Yaskawa INFORM job: DEMO_ROOF_UPPER_0625_3PAINT_54.JBI

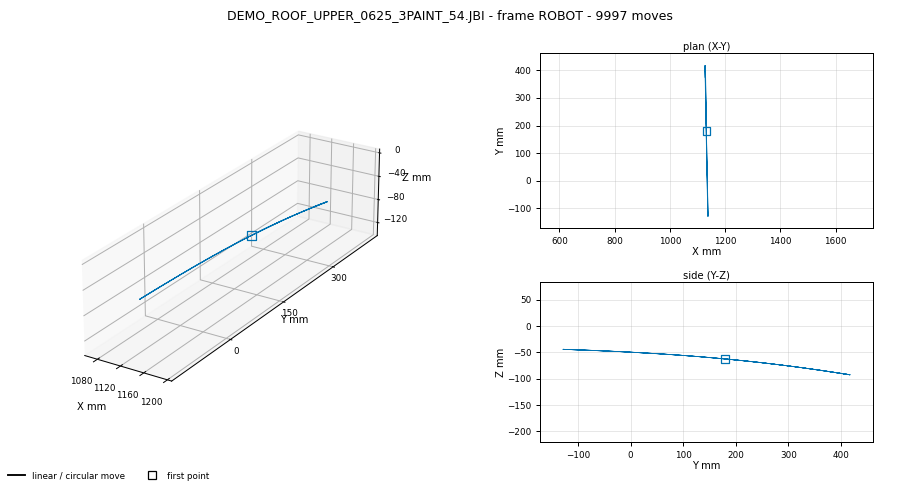
[picture p0: tool path of DEMO_ROOF_UPPER_0625_3PAINT_54.JBI in frame ROBOT, 9997 of 9997 moves have a stored position in this frame; points joined in program order, loops and branches not executed]
/JOB
//NAME DEMO_ROOF_UPPER_0625_3PAINT54
//POS
///NPOS 9997,0,0,0,0,0
///TOOL 0
///USER 0
///POSTYPE ROBOT
///RECTAN
///RCONF 1,0,0,0,0,0,0,0,0,0,0,0,0,0,0,0,0,0,0,0,0,0,0,0
C00000=1132.643,178.804,-62.011,-179.310,9.058,149.575
C00001=1132.639,179.053,-62.034,-179.309,9.060,149.575
C00002=1132.634,179.302,-62.058,-179.306,9.063,149.575
C00003=1132.629,179.551,-62.081,-179.303,9.067,149.575
C00004=1132.624,179.799,-62.104,-179.299,9.071,149.575
C00005=1132.620,180.048,-62.127,-179.296,9.074,149.575
C00006=1132.615,180.297,-62.150,-179.293,9.077,149.575
C00007=1132.611,180.546,-62.174,-179.290,9.081,149.575
C00008=1132.606,180.795,-62.198,-179.287,9.085,149.575
C00009=1132.602,181.044,-62.221,-179.284,9.088,149.575
C00010=1132.597,181.293,-62.244,-179.281,9.092,149.575
C00011=1132.592,181.541,-62.268,-179.278,9.094,149.575
C00012=1132.588,181.790,-62.292,-179.275,9.098,149.575
C00013=1132.583,182.039,-62.315,-179.272,9.101,149.575
C00014=1132.579,182.288,-62.339,-179.268,9.105,149.575
C00015=1132.574,182.537,-62.363,-179.266,9.108,149.575
C00016=1132.569,182.786,-62.386,-179.263,9.111,149.575
C00017=1132.565,183.035,-62.410,-179.260,9.114,149.575
C00018=1132.561,183.284,-62.434,-179.257,9.118,149.575
C00019=1132.556,183.533,-62.457,-179.254,9.120,149.575
C00020=1132.552,183.781,-62.481,-179.251,9.124,149.575
C00021=1132.547,184.030,-62.505,-179.249,9.127,149.575
C00022=1132.542,184.279,-62.528,-179.246,9.130,149.575
C00023=1132.538,184.494,-62.549,-179.244,9.132,149.575
C00024=1132.535,184.707,-62.569,-179.241,9.135,149.575
C00025=1132.531,184.922,-62.589,-179.239,9.138,149.575
C00026=1132.527,185.137,-62.610,-179.237,9.141,149.575
C00027=1132.523,185.351,-62.631,-179.235,9.143,149.575
C00028=1132.519,185.566,-62.651,-179.232,9.146,149.575
C00029=1132.515,185.781,-62.672,-179.230,9.148,149.575
C00030=1132.512,185.995,-62.692,-179.228,9.151,149.575
C00031=1132.506,186.244,-62.716,-179.226,9.154,149.575
C00032=1132.502,186.493,-62.740,-179.223,9.157,149.575
C00033=1132.497,186.741,-62.764,-179.221,9.160,149.575
C00034=1132.493,186.990,-62.787,-179.218,9.163,149.575
C00035=1132.488,187.239,-62.811,-179.215,9.166,149.575
C00036=1132.484,187.487,-62.835,-179.213,9.168,149.575
C00037=1132.479,187.736,-62.859,-179.211,9.171,149.575
C00038=1132.475,187.986,-62.884,-179.208,9.174,149.575
C00039=1132.470,188.235,-62.907,-179.206,9.177,149.575
C00040=1132.466,188.483,-62.931,-179.204,9.180,149.575
C00041=1132.461,188.732,-62.955,-179.202,9.182,149.575
C00042=1132.456,188.981,-62.979,-179.199,9.185,149.575
C00043=1132.451,189.229,-63.003,-179.197,9.188,149.575
C00044=1132.447,189.478,-63.027,-179.195,9.191,149.575
C00045=1132.443,189.727,-63.051,-179.193,9.193,149.575
C00046=1132.438,189.976,-63.075,-179.191,9.196,149.575
C00047=1132.434,190.224,-63.099,-179.189,9.199,149.575
C00048=1132.429,190.474,-63.123,-179.187,9.202,149.575
C00049=1132.424,190.722,-63.147,-179.185,9.204,149.575
C00050=1132.420,190.971,-63.172,-179.183,9.207,149.575
C00051=1132.415,191.220,-63.196,-179.181,9.210,149.576
C00052=1132.411,191.469,-63.220,-179.179,9.212,149.576
C00053=1132.406,191.717,-63.244,-179.177,9.215,149.576
C00054=1132.402,191.966,-63.268,-179.175,9.217,149.576
C00055=1132.397,192.215,-63.293,-179.174,9.220,149.576
C00056=1132.393,192.464,-63.317,-179.172,9.222,149.576
C00057=1132.388,192.713,-63.340,-179.170,9.226,149.576
C00058=1132.383,192.961,-63.365,-179.168,9.228,149.576
C00059=1132.379,193.210,-63.389,-179.166,9.231,149.577
C00060=1132.375,193.459,-63.414,-179.164,9.233,149.577
C00061=1132.370,193.708,-63.438,-179.163,9.236,149.577
C00062=1132.365,193.956,-63.462,-179.161,9.238,149.577
C00063=1132.361,194.205,-63.486,-179.160,9.240,149.577
C00064=1132.356,194.454,-63.511,-179.158,9.242,149.577
C00065=1132.352,194.703,-63.535,-179.157,9.245,149.577
C00066=1132.347,194.951,-63.559,-179.155,9.248,149.578
C00067=1132.343,195.201,-63.584,-179.153,9.250,149.578
C00068=1132.338,195.449,-63.608,-179.152,9.253,149.578
C00069=1132.334,195.698,-63.632,-179.151,9.255,149.578
C00070=1132.329,195.946,-63.657,-179.150,9.257,149.578
C00071=1132.325,196.195,-63.681,-179.148,9.260,149.579
C00072=1132.320,196.444,-63.706,-179.145,9.263,149.578
C00073=1132.316,196.692,-63.730,-179.140,9.268,149.578
C00074=1132.312,196.942,-63.754,-179.136,9.272,149.578
C00075=1132.307,197.190,-63.779,-179.132,9.275,149.578
C00076=1132.302,197.439,-63.803,-179.128,9.279,149.578
C00077=1132.297,197.687,-63.828,-179.124,9.284,149.578
C00078=1132.293,197.937,-63.852,-179.120,9.287,149.577
C00079=1132.289,198.151,-63.873,-179.116,9.291,149.577
C00080=1132.285,198.365,-63.895,-179.112,9.294,149.577
C00081=1132.281,198.580,-63.916,-179.109,9.297,149.577
C00082=1132.277,198.795,-63.937,-179.106,9.300,149.577
C00083=1132.274,199.009,-63.958,-179.103,9.303,149.576
C00084=1132.270,199.223,-63.979,-179.099,9.306,149.576
C00085=1132.265,199.437,-64.001,-179.096,9.309,149.576
C00086=1132.261,199.652,-64.022,-179.093,9.313,149.576
C00087=1132.258,199.901,-64.047,-179.089,9.316,149.576
C00088=1132.253,200.149,-64.071,-179.086,9.320,149.576
C00089=1132.248,200.399,-64.096,-179.082,9.323,149.576
C00090=1132.244,200.647,-64.121,-179.078,9.327,149.576
C00091=1132.239,200.895,-64.146,-179.075,9.330,149.575
C00092=1132.235,201.144,-64.170,-179.071,9.334,149.575
C00093=1132.230,201.393,-64.195,-179.068,9.336,149.575
C00094=1132.226,201.642,-64.221,-179.064,9.340,149.575
C00095=1132.221,201.890,-64.245,-179.061,9.343,149.575
C00096=1132.217,202.140,-64.270,-179.058,9.346,149.574
C00097=1132.212,202.388,-64.295,-179.054,9.349,149.574
C00098=1132.208,202.637,-64.320,-179.051,9.353,149.574
C00099=1132.203,202.886,-64.344,-179.048,9.356,149.574
C00100=1132.199,203.134,-64.370,-179.045,9.358,149.574
C00101=1132.195,203.383,-64.394,-179.041,9.362,149.574
C00102=1132.190,203.632,-64.420,-179.039,9.365,149.574
C00103=1132.185,203.880,-64.445,-179.036,9.368,149.574
C00104=1132.181,204.129,-64.470,-179.032,9.371,149.574
C00105=1132.177,204.378,-64.494,-179.029,9.374,149.573
C00106=1132.172,204.626,-64.520,-179.026,9.377,149.573
C00107=1132.167,204.875,-64.545,-179.023,9.379,149.573
C00108=1132.163,205.124,-64.571,-179.021,9.383,149.573
C00109=1132.159,205.372,-64.595,-179.018,9.385,149.573
C00110=1132.154,205.621,-64.620,-179.015,9.388,149.573
C00111=1132.149,205.870,-64.645,-179.012,9.391,149.573
C00112=1132.145,206.119,-64.671,-179.009,9.394,149.573
C00113=1132.140,206.367,-64.696,-179.006,9.397,149.573
C00114=1132.136,206.616,-64.721,-179.004,9.400,149.573
C00115=1132.132,206.864,-64.746,-179.002,9.402,149.572
C00116=1132.127,207.113,-64.772,-178.999,9.405,149.573
C00117=1132.123,207.362,-64.797,-178.996,9.408,149.573
C00118=1132.118,207.610,-64.822,-178.994,9.410,149.572
C00119=1132.114,207.859,-64.848,-178.992,9.413,149.572
C00120=1132.109,208.108,-64.873,-178.990,9.415,149.573
C00121=1132.104,208.357,-64.898,-178.987,9.418,149.572
C00122=1132.100,208.605,-64.924,-178.985,9.420,149.572
C00123=1132.096,208.854,-64.948,-178.982,9.424,149.572
C00124=1132.092,209.103,-64.974,-178.980,9.426,149.573
C00125=1132.087,209.351,-64.999,-178.979,9.428,149.573
C00126=1132.083,209.600,-65.025,-178.976,9.431,149.573
C00127=1132.078,209.849,-65.050,-178.974,9.434,149.573
C00128=1132.073,210.097,-65.076,-178.972,9.436,149.573
C00129=1132.069,210.346,-65.101,-178.970,9.438,149.573
C00130=1132.065,210.595,-65.127,-178.968,9.441,149.573
C00131=1132.060,210.843,-65.152,-178.967,9.443,149.573
C00132=1132.055,211.092,-65.178,-178.965,9.446,149.573
C00133=1132.051,211.340,-65.203,-178.963,9.448,149.573
C00134=1132.046,211.589,-65.229,-178.961,9.450,149.573
C00135=1132.043,211.803,-65.250,-178.960,9.453,149.573
C00136=1132.039,212.018,-65.273,-178.959,9.455,149.573
C00137=1132.035,212.232,-65.295,-178.957,9.457,149.573
C00138=1132.031,212.446,-65.316,-178.956,9.459,149.574
C00139=1132.027,212.661,-65.338,-178.954,9.462,149.574
C00140=1132.024,212.875,-65.361,-178.953,9.463,149.574
C00141=1132.020,213.089,-65.383,-178.952,9.465,149.574
C00142=1132.015,213.303,-65.405,-178.950,9.467,149.574
C00143=1132.011,213.552,-65.431,-178.949,9.470,149.574
C00144=1132.007,213.801,-65.456,-178.947,9.473,149.575
C00145=1132.002,214.049,-65.482,-178.946,9.475,149.575
C00146=1131.998,214.298,-65.508,-178.944,9.478,149.575
C00147=1131.993,214.547,-65.533,-178.942,9.480,149.575
C00148=1131.989,214.796,-65.558,-178.940,9.484,149.575
C00149=1131.984,215.044,-65.584,-178.938,9.486,149.575
C00150=1131.980,215.293,-65.609,-178.937,9.489,149.576
C00151=1131.976,215.542,-65.635,-178.934,9.492,149.576
C00152=1131.971,215.790,-65.661,-178.933,9.494,149.576
C00153=1131.967,216.039,-65.686,-178.931,9.497,149.576
C00154=1131.962,216.287,-65.712,-178.929,9.500,149.576
C00155=1131.958,216.536,-65.738,-178.927,9.503,149.576
C00156=1131.953,216.784,-65.765,-178.924,9.506,149.576
C00157=1131.949,217.033,-65.790,-178.922,9.509,149.577
C00158=1131.945,217.282,-65.816,-178.920,9.511,149.577
C00159=1131.940,217.530,-65.842,-178.918,9.515,149.577
C00160=1131.935,217.778,-65.867,-178.916,9.518,149.577
C00161=1131.931,218.027,-65.893,-178.914,9.520,149.577
C00162=1131.927,218.276,-65.919,-178.911,9.523,149.577
C00163=1131.922,218.525,-65.945,-178.909,9.527,149.577
C00164=1131.917,218.773,-65.970,-178.907,9.530,149.577
C00165=1131.913,219.022,-65.996,-178.905,9.532,149.577
C00166=1131.909,219.270,-66.023,-178.902,9.535,149.577
C00167=1131.905,219.519,-66.048,-178.900,9.539,149.578
C00168=1131.901,219.768,-66.074,-178.897,9.542,149.578
C00169=1131.895,220.016,-66.100,-178.895,9.545,149.578
C00170=1131.891,220.265,-66.126,-178.892,9.548,149.578
C00171=1131.887,220.513,-66.152,-178.890,9.551,149.578
C00172=1131.883,220.762,-66.178,-178.887,9.554,149.578
C00173=1131.878,221.011,-66.204,-178.884,9.558,149.578
C00174=1131.874,221.260,-66.230,-178.881,9.561,149.578
C00175=1131.869,221.508,-66.256,-178.879,9.564,149.578
C00176=1131.865,221.756,-66.282,-178.876,9.567,149.578
C00177=1131.860,222.005,-66.308,-178.874,9.570,149.578
C00178=1131.856,222.254,-66.335,-178.871,9.574,149.578
C00179=1131.852,222.502,-66.361,-178.868,9.577,149.578
C00180=1131.847,222.752,-66.387,-178.865,9.580,149.578
C00181=1131.843,223.000,-66.413,-178.862,9.584,149.578
C00182=1131.838,223.248,-66.439,-178.859,9.587,149.578
C00183=1131.833,223.497,-66.465,-178.856,9.591,149.578
C00184=1131.829,223.745,-66.492,-178.853,9.594,149.578
C00185=1131.825,223.994,-66.517,-178.850,9.598,149.578
C00186=1131.820,224.242,-66.544,-178.847,9.600,149.578
C00187=1131.816,224.491,-66.570,-178.844,9.604,149.578
C00188=1131.811,224.740,-66.597,-178.840,9.608,149.578
C00189=1131.807,224.989,-66.623,-178.838,9.611,149.578
C00190=1131.803,225.237,-66.649,-178.834,9.614,149.578
C00191=1131.799,225.451,-66.672,-178.832,9.618,149.578
C00192=1131.795,225.665,-66.695,-178.829,9.620,149.578
C00193=1131.791,225.879,-66.717,-178.826,9.623,149.578
C00194=1131.788,226.094,-66.740,-178.823,9.626,149.578
C00195=1131.784,226.308,-66.763,-178.820,9.629,149.578
C00196=1131.780,226.522,-66.786,-178.817,9.633,149.578
C00197=1131.776,226.736,-66.809,-178.814,9.636,149.578
C00198=1131.772,226.951,-66.831,-178.811,9.638,149.578
C00199=1131.768,227.199,-66.858,-178.808,9.642,149.578
C00200=1131.764,227.447,-66.885,-178.804,9.645,149.577
C00201=1131.759,227.696,-66.911,-178.801,9.649,149.577
C00202=1131.755,227.945,-66.937,-178.797,9.652,149.577
C00203=1131.750,228.193,-66.964,-178.793,9.656,149.577
C00204=1131.746,228.441,-66.991,-178.790,9.659,149.577
C00205=1131.741,228.690,-67.017,-178.786,9.663,149.577
C00206=1131.737,228.939,-67.044,-178.783,9.666,149.577
C00207=1131.733,229.187,-67.071,-178.779,9.670,149.577
C00208=1131.728,229.436,-67.098,-178.775,9.673,149.576
C00209=1131.724,229.684,-67.124,-178.771,9.677,149.576
C00210=1131.719,229.933,-67.151,-178.767,9.681,149.576
C00211=1131.715,230.181,-67.178,-178.763,9.684,149.576
C00212=1131.711,230.430,-67.204,-178.760,9.688,149.576
C00213=1131.706,230.678,-67.231,-178.756,9.691,149.576
C00214=1131.701,230.927,-67.258,-178.752,9.694,149.575
C00215=1131.697,231.175,-67.285,-178.749,9.698,149.575
C00216=1131.693,231.423,-67.312,-178.745,9.701,149.575
C00217=1131.688,231.672,-67.339,-178.741,9.704,149.575
C00218=1131.684,231.921,-67.365,-178.737,9.708,149.575
C00219=1131.680,232.170,-67.392,-178.734,9.711,149.574
C00220=1131.675,232.418,-67.419,-178.731,9.714,149.574
C00221=1131.670,232.667,-67.446,-178.727,9.718,149.574
C00222=1131.667,232.915,-67.473,-178.724,9.720,149.574
C00223=1131.662,233.163,-67.500,-178.720,9.724,149.574
C00224=1131.658,233.411,-67.528,-178.717,9.726,149.574
C00225=1131.654,233.660,-67.555,-178.714,9.729,149.573
C00226=1131.650,233.909,-67.581,-178.711,9.733,149.573
C00227=1131.645,234.157,-67.609,-178.708,9.735,149.573
C00228=1131.640,234.406,-67.636,-178.705,9.738,149.573
C00229=1131.636,234.654,-67.663,-178.701,9.741,149.573
C00230=1131.631,234.903,-67.690,-178.698,9.744,149.573
C00231=1131.627,235.152,-67.717,-178.695,9.747,149.573
C00232=1131.623,235.399,-67.744,-178.692,9.750,149.572
C00233=1131.619,235.648,-67.771,-178.689,9.752,149.572
C00234=1131.614,235.896,-67.798,-178.686,9.755,149.572
C00235=1131.610,236.146,-67.826,-178.683,9.758,149.572
C00236=1131.605,236.394,-67.853,-178.680,9.761,149.572
C00237=1131.601,236.642,-67.881,-178.678,9.764,149.572
C00238=1131.596,236.890,-67.908,-178.675,9.766,149.572
C00239=1131.592,237.139,-67.935,-178.672,9.769,149.572
C00240=1131.589,237.387,-67.962,-178.670,9.771,149.572
C00241=1131.584,237.636,-67.989,-178.667,9.774,149.571
C00242=1131.579,237.884,-68.016,-178.664,9.777,149.571
C00243=1131.575,238.133,-68.044,-178.662,9.779,149.571
C00244=1131.571,238.381,-68.072,-178.659,9.782,149.571
C00245=1131.566,238.630,-68.099,-178.657,9.784,149.571
C00246=1131.562,238.878,-68.126,-178.654,9.787,149.571
C00247=1131.558,239.092,-68.150,-178.652,9.789,149.571
C00248=1131.554,239.307,-68.173,-178.650,9.791,149.571
C00249=1131.551,239.520,-68.197,-178.647,9.793,149.571
C00250=1131.546,239.734,-68.221,-178.646,9.795,149.571
C00251=1131.543,239.948,-68.245,-178.644,9.797,149.571
C00252=1131.539,240.163,-68.268,-178.642,9.799,149.571
C00253=1131.536,240.377,-68.292,-178.640,9.801,149.571
C00254=1131.531,240.590,-68.316,-178.638,9.803,149.571
C00255=1131.527,240.839,-68.344,-178.636,9.806,149.571
C00256=1131.523,241.088,-68.371,-178.634,9.808,149.571
C00257=1131.518,241.335,-68.399,-178.632,9.810,149.571
C00258=1131.514,241.585,-68.426,-178.630,9.812,149.571
C00259=1131.510,241.832,-68.454,-178.628,9.815,149.571
C00260=1131.505,242.081,-68.481,-178.626,9.817,149.571
C00261=1131.502,242.330,-68.509,-178.624,9.819,149.571
C00262=1131.497,242.578,-68.536,-178.622,9.821,149.571
C00263=1131.493,242.826,-68.564,-178.620,9.824,149.571
C00264=1131.488,243.075,-68.591,-178.618,9.826,149.571
C00265=1131.484,243.323,-68.619,-178.617,9.827,149.571
C00266=1131.479,243.572,-68.646,-178.615,9.830,149.571
C00267=1131.476,243.820,-68.674,-178.613,9.832,149.571
C00268=1131.470,244.069,-68.702,-178.611,9.835,149.571
C00269=1131.466,244.317,-68.730,-178.610,9.836,149.571
C00270=1131.462,244.565,-68.758,-178.608,9.839,149.572
C00271=1131.458,244.814,-68.785,-178.607,9.841,149.572
C00272=1131.454,245.062,-68.813,-178.606,9.843,149.572
C00273=1131.449,245.311,-68.840,-178.604,9.844,149.572
C00274=1131.445,245.559,-68.868,-178.603,9.847,149.572
C00275=1131.441,245.807,-68.896,-178.602,9.849,149.572
C00276=1131.436,246.056,-68.924,-178.601,9.851,149.572
C00277=1131.431,246.304,-68.951,-178.599,9.853,149.573
C00278=1131.428,246.553,-68.980,-178.598,9.855,149.573
C00279=1131.423,246.801,-69.007,-178.597,9.857,149.573
C00280=1131.419,247.050,-69.035,-178.596,9.859,149.573
C00281=1131.415,247.298,-69.063,-178.595,9.861,149.573
C00282=1131.409,247.546,-69.090,-178.590,9.865,149.573
C00283=1131.406,247.795,-69.118,-178.583,9.871,149.573
C00284=1131.401,248.043,-69.146,-178.575,9.876,149.572
C00285=1131.398,248.291,-69.174,-178.568,9.882,149.571
C00286=1131.392,248.540,-69.202,-178.561,9.888,149.571
C00287=1131.388,248.789,-69.230,-178.554,9.893,149.570
C00288=1131.384,249.037,-69.258,-178.548,9.897,149.570
C00289=1131.380,249.286,-69.287,-178.542,9.902,149.569
C00290=1131.375,249.533,-69.314,-178.536,9.906,149.569
C00291=1131.371,249.782,-69.342,-178.531,9.911,149.568
C00292=1131.366,250.030,-69.371,-178.526,9.914,149.568
C00293=1131.363,250.279,-69.399,-178.520,9.919,149.567
C00294=1131.358,250.527,-69.427,-178.516,9.922,149.567
C00295=1131.354,250.776,-69.456,-178.511,9.925,149.567
C00296=1131.349,251.023,-69.483,-178.507,9.928,149.566
C00297=1131.345,251.272,-69.512,-178.503,9.932,149.566
C00298=1131.341,251.520,-69.540,-178.499,9.935,149.566
C00299=1131.337,251.769,-69.568,-178.496,9.938,149.566
C00300=1131.332,252.018,-69.597,-178.493,9.940,149.565
C00301=1131.328,252.266,-69.624,-178.490,9.943,149.565
C00302=1131.324,252.514,-69.654,-178.487,9.945,149.565
C00303=1131.320,252.728,-69.678,-178.485,9.947,149.565
C00304=1131.316,252.942,-69.703,-178.483,9.949,149.565
C00305=1131.313,253.156,-69.727,-178.482,9.950,149.565
C00306=1131.309,253.370,-69.751,-178.480,9.952,149.565
C00307=1131.305,253.584,-69.776,-178.479,9.953,149.565
C00308=1131.301,253.798,-69.800,-178.477,9.954,149.565
C00309=1131.298,254.011,-69.825,-178.477,9.956,149.565
C00310=1131.294,254.225,-69.850,-178.476,9.956,149.565
C00311=1131.290,254.473,-69.878,-178.476,9.958,149.565
C00312=1131.285,254.722,-69.906,-178.475,9.959,149.565
C00313=1131.281,254.971,-69.934,-178.476,9.960,149.566
C00314=1131.277,255.218,-69.963,-178.476,9.960,149.566
C00315=1131.273,255.467,-69.992,-178.476,9.962,149.566
C00316=1131.268,255.716,-70.020,-178.478,9.962,149.567
C00317=1131.264,255.963,-70.048,-178.479,9.962,149.567
C00318=1131.259,256.212,-70.077,-178.476,9.965,149.567
C00319=1131.255,256.460,-70.105,-178.473,9.968,149.567
C00320=1131.251,256.708,-70.134,-178.469,9.971,149.567
C00321=1131.247,256.957,-70.162,-178.466,9.974,149.567
C00322=1131.242,257.205,-70.191,-178.463,9.977,149.566
C00323=1131.238,257.454,-70.220,-178.460,9.980,149.566
C00324=1131.234,257.702,-70.248,-178.457,9.982,149.566
C00325=1131.229,257.950,-70.277,-178.455,9.985,149.566
C00326=1131.226,258.198,-70.305,-178.451,9.989,149.566
C00327=1131.221,258.447,-70.334,-178.448,9.991,149.566
C00328=1131.216,258.695,-70.363,-178.445,9.994,149.566
C00329=1131.213,258.943,-70.391,-178.442,9.998,149.566
C00330=1131.208,259.192,-70.420,-178.439,10.000,149.566
C00331=1131.204,259.439,-70.449,-178.435,10.004,149.566
C00332=1131.200,259.688,-70.477,-178.432,10.007,149.565
C00333=1131.195,259.937,-70.507,-178.429,10.009,149.565
C00334=1131.191,260.184,-70.535,-178.425,10.013,149.565
C00335=1131.187,260.433,-70.563,-178.422,10.016,149.565
C00336=1131.182,260.682,-70.593,-178.418,10.019,149.565
C00337=1131.178,260.930,-70.622,-178.415,10.022,149.565
C00338=1131.174,261.178,-70.650,-178.412,10.025,149.564
C00339=1131.169,261.427,-70.679,-178.408,10.028,149.564
C00340=1131.165,261.675,-70.708,-178.404,10.032,149.564
C00341=1131.162,261.923,-70.737,-178.400,10.035,149.564
C00342=1131.157,262.171,-70.765,-178.397,10.037,149.563
C00343=1131.152,262.419,-70.795,-178.393,10.041,149.563
C00344=1131.148,262.668,-70.824,-178.389,10.044,149.563
C00345=1131.144,262.916,-70.853,-178.385,10.047,149.563
C00346=1131.140,263.164,-70.882,-178.382,10.051,149.563
C00347=1131.135,263.413,-70.910,-178.378,10.054,149.562
C00348=1131.131,263.661,-70.940,-178.374,10.057,149.562
C00349=1131.127,263.909,-70.969,-178.370,10.060,149.562
C00350=1131.122,264.158,-70.998,-178.366,10.063,149.562
C00351=1131.118,264.406,-71.027,-178.362,10.066,149.561
C00352=1131.113,264.654,-71.057,-178.359,10.068,149.561
C00353=1131.110,264.902,-71.085,-178.357,10.070,149.561
C00354=1131.106,265.150,-71.115,-178.355,10.074,149.561
C00355=1131.101,265.399,-71.144,-178.352,10.076,149.561
C00356=1131.097,265.647,-71.173,-178.350,10.078,149.561
C00357=1131.093,265.896,-71.202,-178.347,10.080,149.561
C00358=1131.088,266.143,-71.232,-178.345,10.082,149.561
C00359=1131.085,266.358,-71.256,-178.343,10.085,149.561
C00360=1131.081,266.571,-71.282,-178.340,10.087,149.561
C00361=1131.077,266.785,-71.307,-178.338,10.089,149.560
C00362=1131.074,266.998,-71.333,-178.336,10.091,149.560
C00363=1131.070,267.212,-71.357,-178.334,10.093,149.560
C00364=1131.067,267.427,-71.383,-178.332,10.095,149.560
C00365=1131.063,267.640,-71.408,-178.329,10.097,149.560
C00366=1131.059,267.854,-71.434,-178.327,10.099,149.560
C00367=1131.055,268.102,-71.463,-178.324,10.102,149.560
C00368=1131.050,268.350,-71.492,-178.322,10.104,149.560
C00369=1131.046,268.599,-71.522,-178.319,10.107,149.560
C00370=1131.042,268.847,-71.551,-178.317,10.109,149.560
C00371=1131.038,269.095,-71.581,-178.314,10.111,149.560
C00372=1131.034,269.343,-71.610,-178.311,10.114,149.560
C00373=1131.029,269.591,-71.639,-178.309,10.116,149.559
C00374=1131.025,269.839,-71.669,-178.306,10.119,149.559
C00375=1131.021,270.087,-71.698,-178.303,10.122,149.559
C00376=1131.016,270.336,-71.728,-178.300,10.124,149.559
C00377=1131.012,270.584,-71.757,-178.298,10.126,149.559
C00378=1131.008,270.832,-71.787,-178.295,10.129,149.559
C00379=1131.004,271.081,-71.816,-178.292,10.132,149.559
C00380=1131.000,271.329,-71.846,-178.289,10.135,149.559
C00381=1130.995,271.577,-71.875,-178.286,10.137,149.559
C00382=1130.991,271.825,-71.904,-178.284,10.139,149.558
C00383=1130.987,272.074,-71.934,-178.281,10.142,149.558
C00384=1130.982,272.322,-71.964,-178.278,10.145,149.558
C00385=1130.978,272.570,-71.994,-178.274,10.147,149.558
C00386=1130.974,272.818,-72.024,-178.271,10.150,149.558
C00387=1130.970,273.066,-72.053,-178.268,10.153,149.558
C00388=1130.966,273.315,-72.082,-178.266,10.156,149.558
C00389=1130.962,273.563,-72.112,-178.263,10.158,149.558
C00390=1130.958,273.811,-72.142,-178.260,10.161,149.557
C00391=1130.953,274.059,-72.172,-178.257,10.164,149.557
C00392=1130.949,274.307,-72.202,-178.253,10.166,149.557
C00393=1130.944,274.556,-72.231,-178.250,10.169,149.557
C00394=1130.941,274.803,-72.261,-178.248,10.172,149.557
C00395=1130.936,275.052,-72.291,-178.245,10.175,149.557
C00396=1130.931,275.300,-72.321,-178.241,10.177,149.556
C00397=1130.928,275.548,-72.351,-178.238,10.180,149.556
C00398=1130.923,275.796,-72.380,-178.235,10.183,149.556
C00399=1130.919,276.044,-72.410,-178.231,10.186,149.556
C00400=1130.915,276.293,-72.441,-178.228,10.188,149.556
C00401=1130.911,276.541,-72.470,-178.225,10.191,149.556
C00402=1130.907,276.790,-72.500,-178.222,10.194,149.556
C00403=1130.903,277.037,-72.530,-178.219,10.197,149.555
C00404=1130.898,277.286,-72.560,-178.215,10.200,149.555
C00405=1130.894,277.533,-72.590,-178.212,10.202,149.555
C00406=1130.890,277.782,-72.620,-178.208,10.205,149.555
C00407=1130.885,278.030,-72.650,-178.205,10.208,149.555
C00408=1130.881,278.278,-72.680,-178.202,10.211,149.554
C00409=1130.878,278.526,-72.710,-178.198,10.214,149.554
C00410=1130.873,278.775,-72.740,-178.195,10.217,149.554
C00411=1130.869,279.022,-72.771,-178.192,10.219,149.554
C00412=1130.865,279.271,-72.800,-178.188,10.223,149.554
C00413=1130.860,279.519,-72.831,-178.185,10.225,149.553
C00414=1130.856,279.767,-72.860,-178.181,10.229,149.553
C00415=1130.853,279.981,-72.887,-178.179,10.230,149.553
C00416=1130.849,280.194,-72.912,-178.176,10.233,149.553
C00417=1130.846,280.408,-72.939,-178.172,10.235,149.553
C00418=1130.841,280.622,-72.965,-178.169,10.238,149.553
C00419=1130.838,280.835,-72.991,-178.166,10.240,149.552
C00420=1130.835,281.049,-73.017,-178.163,10.243,149.552
C00421=1130.831,281.262,-73.043,-178.160,10.246,149.552
C00422=1130.828,281.476,-73.069,-178.157,10.247,149.552
C00423=1130.823,281.724,-73.100,-178.154,10.250,149.551
C00424=1130.819,281.972,-73.129,-178.151,10.253,149.551
C00425=1130.814,282.220,-73.160,-178.148,10.255,149.551
C00426=1130.811,282.469,-73.191,-178.145,10.258,149.551
C00427=1130.806,282.717,-73.221,-178.141,10.260,149.551
C00428=1130.802,282.965,-73.251,-178.139,10.263,149.551
C00429=1130.797,283.213,-73.282,-178.135,10.266,149.550
C00430=1130.794,283.461,-73.312,-178.132,10.268,149.550
C00431=1130.790,283.709,-73.343,-178.129,10.271,149.550
C00432=1130.786,283.957,-73.373,-178.126,10.274,149.550
C00433=1130.781,284.205,-73.404,-178.124,10.276,149.550
C00434=1130.777,284.454,-73.434,-178.120,10.278,149.549
C00435=1130.773,284.702,-73.464,-178.117,10.281,149.549
C00436=1130.768,284.950,-73.495,-178.114,10.283,149.549
C00437=1130.764,285.197,-73.525,-178.111,10.286,149.549
C00438=1130.760,285.446,-73.556,-178.108,10.289,149.549
C00439=1130.756,285.694,-73.587,-178.105,10.291,149.549
C00440=1130.752,285.942,-73.617,-178.102,10.294,149.549
C00441=1130.748,286.190,-73.648,-178.099,10.296,149.548
C00442=1130.743,286.438,-73.679,-178.096,10.299,149.548
C00443=1130.739,286.686,-73.709,-178.093,10.301,149.548
C00444=1130.735,286.934,-73.740,-178.090,10.303,149.548
C00445=1130.731,287.183,-73.771,-178.087,10.306,149.547
C00446=1130.727,287.430,-73.801,-178.084,10.309,149.547
C00447=1130.722,287.678,-73.832,-178.081,10.311,149.547
C00448=1130.718,287.927,-73.863,-178.077,10.314,149.547
C00449=1130.714,288.174,-73.894,-178.074,10.317,149.547
C00450=1130.710,288.422,-73.924,-178.071,10.319,149.547
C00451=1130.706,288.671,-73.955,-178.068,10.322,149.547
C00452=1130.702,288.919,-73.986,-178.065,10.324,149.546
C00453=1130.698,289.167,-74.017,-178.062,10.327,149.546
C00454=1130.694,289.415,-74.048,-178.059,10.329,149.546
C00455=1130.689,289.663,-74.079,-178.056,10.331,149.546
C00456=1130.686,289.911,-74.110,-178.053,10.334,149.546
C00457=1130.681,290.159,-74.140,-178.050,10.336,149.545
C00458=1130.677,290.408,-74.171,-178.047,10.339,149.545
C00459=1130.673,290.655,-74.203,-178.044,10.342,149.545
C00460=1130.668,290.903,-74.234,-178.041,10.344,149.545
C00461=1130.665,291.151,-74.264,-178.037,10.347,149.545
C00462=1130.660,291.399,-74.295,-178.035,10.350,149.545
C00463=1130.656,291.648,-74.326,-178.031,10.352,149.544
C00464=1130.652,291.895,-74.358,-178.028,10.355,149.544
C00465=1130.647,292.143,-74.388,-178.025,10.357,149.544
C00466=1130.643,292.392,-74.419,-178.023,10.359,149.544
C00467=1130.640,292.639,-74.450,-178.019,10.362,149.544
C00468=1130.636,292.888,-74.481,-178.016,10.364,149.543
C00469=1130.631,293.135,-74.512,-178.013,10.367,149.543
C00470=1130.627,293.384,-74.544,-178.010,10.370,149.543
C00471=1130.623,293.597,-74.571,-178.007,10.372,149.543
C00472=1130.620,293.810,-74.597,-178.004,10.374,149.543
C00473=1130.617,294.024,-74.624,-178.002,10.376,149.543
C00474=1130.613,294.237,-74.651,-177.999,10.379,149.543
C00475=1130.609,294.451,-74.678,-177.996,10.380,149.542
C00476=1130.606,294.664,-74.705,-177.994,10.382,149.542
C00477=1130.602,294.877,-74.732,-177.991,10.385,149.542
C00478=1130.599,295.091,-74.759,-177.989,10.387,149.542
C00479=1130.595,295.340,-74.790,-177.986,10.390,149.542
C00480=1130.590,295.587,-74.821,-177.983,10.392,149.542
C00481=1130.586,295.836,-74.852,-177.979,10.395,149.541
C00482=1130.582,296.083,-74.884,-177.976,10.398,149.541
C00483=1130.578,296.332,-74.915,-177.973,10.400,149.541
C00484=1130.574,296.579,-74.946,-177.970,10.403,149.541
C00485=1130.570,296.827,-74.978,-177.967,10.405,149.541
C00486=1130.565,297.075,-75.009,-177.964,10.408,149.541
C00487=1130.562,297.323,-75.041,-177.961,10.410,149.540
C00488=1130.557,297.571,-75.072,-177.958,10.412,149.540
C00489=1130.553,297.819,-75.103,-177.955,10.415,149.540
C00490=1130.550,298.067,-75.135,-177.952,10.418,149.540
C00491=1130.545,298.315,-75.166,-177.949,10.420,149.540
C00492=1130.541,298.563,-75.198,-177.946,10.423,149.539
C00493=1130.537,298.811,-75.229,-177.942,10.425,149.539
C00494=1130.532,299.060,-75.261,-177.939,10.428,149.539
C00495=1130.528,299.307,-75.293,-177.936,10.430,149.539
C00496=1130.524,299.555,-75.324,-177.933,10.433,149.539
C00497=1130.520,299.804,-75.356,-177.930,10.436,149.538
C00498=1130.516,300.051,-75.387,-177.927,10.438,149.538
C00499=1130.512,300.299,-75.419,-177.924,10.441,149.538
C00500=1130.508,300.546,-75.450,-177.921,10.443,149.538
C00501=1130.504,300.795,-75.481,-177.918,10.445,149.538
C00502=1130.500,301.043,-75.514,-177.915,10.448,149.538
C00503=1130.495,301.291,-75.545,-177.912,10.450,149.537
C00504=1130.492,301.539,-75.577,-177.908,10.453,149.537
C00505=1130.488,301.787,-75.609,-177.905,10.456,149.537
C00506=1130.484,302.034,-75.641,-177.902,10.458,149.537
C00507=1130.479,302.283,-75.672,-177.899,10.461,149.537
C00508=1130.474,302.530,-75.704,-177.896,10.463,149.536
C00509=1130.471,302.779,-75.736,-177.893,10.466,149.536
C00510=1130.467,303.027,-75.767,-177.890,10.468,149.536
C00511=1130.462,303.274,-75.800,-177.887,10.471,149.536
C00512=1130.458,303.522,-75.831,-177.883,10.474,149.536
C00513=1130.455,303.770,-75.863,-177.880,10.476,149.536
C00514=1130.450,304.018,-75.895,-177.878,10.478,149.535
C00515=1130.446,304.266,-75.927,-177.875,10.481,149.535
C00516=1130.442,304.514,-75.959,-177.871,10.483,149.535
C00517=1130.438,304.762,-75.991,-177.868,10.486,149.535
C00518=1130.433,305.010,-76.023,-177.865,10.488,149.535
C00519=1130.430,305.258,-76.055,-177.862,10.491,149.534
C00520=1130.426,305.506,-76.087,-177.859,10.494,149.534
C00521=1130.421,305.753,-76.119,-177.855,10.496,149.534
C00522=1130.417,306.001,-76.151,-177.853,10.499,149.534
C00523=1130.414,306.250,-76.182,-177.849,10.501,149.534
C00524=1130.409,306.498,-76.215,-177.846,10.504,149.534
C00525=1130.405,306.745,-76.246,-177.843,10.506,149.533
C00526=1130.401,306.993,-76.279,-177.840,10.509,149.533
C00527=1130.397,307.207,-76.306,-177.837,10.511,149.533
C00528=1130.394,307.420,-76.334,-177.835,10.513,149.533
C00529=1130.390,307.633,-76.362,-177.832,10.516,149.533
C00530=1130.387,307.847,-76.390,-177.829,10.517,149.533
C00531=1130.383,308.059,-76.417,-177.826,10.520,149.532
C00532=1130.379,308.273,-76.444,-177.824,10.522,149.532
C00533=1130.376,308.487,-76.472,-177.821,10.524,149.532
C00534=1130.372,308.700,-76.500,-177.819,10.526,149.532
C00535=1130.368,308.948,-76.532,-177.815,10.529,149.532
C00536=1130.365,309.196,-76.565,-177.812,10.532,149.532
C00537=1130.361,309.444,-76.597,-177.809,10.534,149.531
C00538=1130.356,309.691,-76.629,-177.806,10.536,149.531
C00539=1130.352,309.939,-76.662,-177.803,10.538,149.531
C00540=1130.348,310.187,-76.694,-177.800,10.541,149.531
C00541=1130.344,310.435,-76.726,-177.797,10.544,149.531
C00542=1130.340,310.683,-76.759,-177.794,10.546,149.530
C00543=1130.336,310.931,-76.791,-177.791,10.549,149.530
C00544=1130.331,311.179,-76.823,-177.787,10.551,149.530
C00545=1130.327,311.426,-76.856,-177.784,10.554,149.530
C00546=1130.324,311.674,-76.888,-177.781,10.557,149.530
C00547=1130.319,311.923,-76.920,-177.778,10.559,149.529
C00548=1130.316,312.170,-76.953,-177.775,10.562,149.529
C00549=1130.311,312.419,-76.985,-177.772,10.564,149.529
C00550=1130.308,312.666,-77.018,-177.768,10.567,149.529
C00551=1130.303,312.914,-77.050,-177.765,10.569,149.529
C00552=1130.299,313.161,-77.083,-177.762,10.572,149.529
C00553=1130.295,313.409,-77.115,-177.759,10.575,149.529
C00554=1130.291,313.657,-77.148,-177.756,10.577,149.528
C00555=1130.287,313.905,-77.180,-177.752,10.579,149.528
C00556=1130.283,314.153,-77.213,-177.750,10.581,149.528
C00557=1130.279,314.401,-77.246,-177.747,10.584,149.528
C00558=1130.275,314.649,-77.278,-177.744,10.587,149.528
C00559=1130.271,314.896,-77.311,-177.741,10.589,149.527
C00560=1130.267,315.145,-77.344,-177.737,10.592,149.527
C00561=1130.263,315.392,-77.376,-177.734,10.594,149.527
C00562=1130.259,315.640,-77.409,-177.731,10.597,149.527
C00563=1130.255,315.888,-77.442,-177.728,10.600,149.527
C00564=1130.251,316.135,-77.474,-177.725,10.602,149.526
C00565=1130.246,316.383,-77.506,-177.721,10.604,149.526
C00566=1130.242,316.631,-77.540,-177.718,10.607,149.526
C00567=1130.239,316.878,-77.572,-177.715,10.610,149.526
C00568=1130.235,317.126,-77.605,-177.712,10.612,149.526
C00569=1130.230,317.375,-77.638,-177.709,10.615,149.525
C00570=1130.226,317.622,-77.671,-177.706,10.617,149.525
C00571=1130.223,317.870,-77.704,-177.703,10.620,149.525
C00572=1130.218,318.117,-77.737,-177.699,10.623,149.525
C00573=1130.214,318.366,-77.769,-177.696,10.625,149.525
C00574=1130.210,318.613,-77.802,-177.694,10.627,149.525
C00575=1130.206,318.861,-77.835,-177.690,10.629,149.524
C00576=1130.202,319.109,-77.868,-177.687,10.632,149.524
C00577=1130.198,319.356,-77.901,-177.684,10.635,149.524
C00578=1130.194,319.604,-77.934,-177.681,10.637,149.524
C00579=1130.190,319.853,-77.967,-177.677,10.639,149.523
C00580=1130.186,320.101,-78.000,-177.675,10.642,149.523
C00581=1130.183,320.348,-78.033,-177.671,10.645,149.523
C00582=1130.178,320.596,-78.066,-177.668,10.647,149.523
C00583=1130.175,320.809,-78.095,-177.666,10.649,149.523
C00584=1130.171,321.022,-78.123,-177.663,10.652,149.523
C00585=1130.168,321.235,-78.152,-177.660,10.654,149.522
C00586=1130.165,321.448,-78.179,-177.657,10.656,149.522
C00587=1130.161,321.661,-78.208,-177.654,10.658,149.522
C00588=1130.157,321.875,-78.237,-177.652,10.660,149.522
C00589=1130.154,322.088,-78.266,-177.649,10.663,149.522
C00590=1130.150,322.302,-78.294,-177.646,10.664,149.522
C00591=1130.146,322.550,-78.327,-177.643,10.667,149.521
C00592=1130.142,322.797,-78.360,-177.640,10.670,149.521
C00593=1130.138,323.045,-78.394,-177.637,10.672,149.521
C00594=1130.135,323.292,-78.427,-177.634,10.675,149.521
C00595=1130.131,323.540,-78.460,-177.631,10.677,149.521
C00596=1130.127,323.787,-78.493,-177.627,10.680,149.521
C00597=1130.123,324.036,-78.527,-177.624,10.682,149.520
C00598=1130.119,324.284,-78.560,-177.621,10.685,149.520
C00599=1130.115,324.531,-78.593,-177.618,10.687,149.520
C00600=1130.111,324.779,-78.626,-177.614,10.690,149.520
C00601=1130.107,325.026,-78.660,-177.611,10.693,149.520
C00602=1130.103,325.274,-78.693,-177.608,10.695,149.519
C00603=1130.099,325.522,-78.726,-177.605,10.698,149.519
C00604=1130.094,325.770,-78.760,-177.602,10.700,149.519
C00605=1130.090,326.018,-78.793,-177.599,10.703,149.519
C00606=1130.086,326.265,-78.827,-177.595,10.705,149.519
C00607=1130.082,326.513,-78.860,-177.593,10.707,149.519
C00608=1130.078,326.761,-78.894,-177.590,10.710,149.518
C00609=1130.075,327.009,-78.927,-177.586,10.712,149.518
C00610=1130.071,327.256,-78.961,-177.583,10.715,149.518
C00611=1130.067,327.504,-78.994,-177.580,10.717,149.518
C00612=1130.062,327.752,-79.027,-177.577,10.720,149.517
C00613=1130.059,327.999,-79.061,-177.573,10.722,149.517
C00614=1130.054,328.247,-79.095,-177.571,10.725,149.517
C00615=1130.050,328.495,-79.128,-177.567,10.727,149.517
C00616=1130.046,328.742,-79.162,-177.564,10.730,149.517
C00617=1130.042,328.990,-79.196,-177.561,10.732,149.516
C00618=1130.038,329.237,-79.229,-177.558,10.735,149.516
C00619=1130.035,329.486,-79.263,-177.554,10.738,149.516
C00620=1130.030,329.733,-79.297,-177.551,10.740,149.516
C00621=1130.026,329.981,-79.331,-177.548,10.743,149.516
C00622=1130.022,330.228,-79.364,-177.545,10.745,149.516
C00623=1130.019,330.476,-79.398,-177.541,10.748,149.515
C00624=1130.015,330.724,-79.431,-177.538,10.750,149.515
C00625=1130.010,330.971,-79.466,-177.535,10.753,149.515
C00626=1130.007,331.219,-79.500,-177.532,10.755,149.515
C00627=1130.003,331.467,-79.533,-177.529,10.758,149.515
C00628=1129.999,331.714,-79.567,-177.525,10.760,149.514
C00629=1129.994,331.962,-79.601,-177.522,10.763,149.514
C00630=1129.991,332.210,-79.635,-177.520,10.765,149.514
C00631=1129.987,332.458,-79.668,-177.516,10.767,149.514
C00632=1129.982,332.705,-79.702,-177.513,10.770,149.514
C00633=1129.979,332.953,-79.737,-177.510,10.772,149.513
C00634=1129.975,333.201,-79.770,-177.507,10.775,149.513
C00635=1129.971,333.448,-79.804,-177.503,10.777,149.513
C00636=1129.967,333.696,-79.839,-177.500,10.780,149.513
C00637=1129.963,333.944,-79.872,-177.497,10.783,149.513
C00638=1129.959,334.191,-79.906,-177.494,10.785,149.512
C00639=1129.955,334.405,-79.935,-177.491,10.787,149.512
C00640=1129.952,334.617,-79.964,-177.488,10.789,149.512
C00641=1129.948,334.830,-79.994,-177.486,10.791,149.512
C00642=1129.946,335.043,-80.023,-177.483,10.794,149.512
C00643=1129.941,335.256,-80.053,-177.480,10.796,149.512
C00644=1129.938,335.469,-80.081,-177.477,10.798,149.511
C00645=1129.935,335.682,-80.111,-177.474,10.800,149.511
C00646=1129.932,335.895,-80.140,-177.472,10.802,149.511
C00647=1129.928,336.143,-80.175,-177.469,10.804,149.511
C00648=1129.924,336.391,-80.208,-177.465,10.807,149.511
C00649=1129.919,336.638,-80.243,-177.462,10.810,149.511
C00650=1129.916,336.886,-80.277,-177.459,10.812,149.510
C00651=1129.912,337.133,-80.311,-177.456,10.815,149.510
C00652=1129.908,337.382,-80.346,-177.453,10.817,149.510
C00653=1129.904,337.629,-80.380,-177.449,10.819,149.510
C00654=1129.900,337.877,-80.414,-177.446,10.822,149.510
C00655=1129.896,338.124,-80.448,-177.443,10.825,149.509
C00656=1129.892,338.371,-80.483,-177.440,10.827,149.509
C00657=1129.889,338.619,-80.517,-177.436,10.830,149.509
C00658=1129.884,338.867,-80.551,-177.433,10.832,149.509
C00659=1129.881,339.114,-80.586,-177.430,10.835,149.509
C00660=1129.876,339.362,-80.620,-177.427,10.837,149.508
C00661=1129.872,339.610,-80.655,-177.423,10.840,149.508
C00662=1129.868,339.857,-80.689,-177.420,10.842,149.508
C00663=1129.864,340.105,-80.724,-177.417,10.845,149.508
C00664=1129.861,340.352,-80.758,-177.414,10.847,149.508
C00665=1129.856,340.600,-80.792,-177.411,10.850,149.507
C00666=1129.853,340.847,-80.826,-177.407,10.852,149.507
C00667=1129.848,341.095,-80.861,-177.404,10.855,149.507
C00668=1129.844,341.343,-80.896,-177.401,10.857,149.507
C00669=1129.840,341.590,-80.929,-177.398,10.860,149.507
C00670=1129.836,341.838,-80.964,-177.395,10.862,149.506
C00671=1129.832,342.085,-80.999,-177.392,10.864,149.506
C00672=1129.829,342.333,-81.034,-177.388,10.867,149.506
C00673=1129.824,342.580,-81.068,-177.385,10.869,149.506
C00674=1129.820,342.828,-81.103,-177.382,10.872,149.505
C00675=1129.817,343.076,-81.137,-177.379,10.874,149.505
C00676=1129.813,343.323,-81.172,-177.376,10.877,149.505
C00677=1129.809,343.571,-81.207,-177.372,10.879,149.505
C00678=1129.805,343.818,-81.241,-177.369,10.882,149.505
C00679=1129.801,344.066,-81.276,-177.366,10.884,149.504
C00680=1129.797,344.313,-81.311,-177.362,10.887,149.504
C00681=1129.793,344.561,-81.346,-177.359,10.889,149.504
C00682=1129.789,344.808,-81.380,-177.356,10.892,149.504
C00683=1129.785,345.056,-81.415,-177.353,10.894,149.504
C00684=1129.781,345.304,-81.450,-177.349,10.897,149.503
C00685=1129.777,345.551,-81.485,-177.346,10.899,149.503
C00686=1129.774,345.799,-81.520,-177.343,10.902,149.503
C00687=1129.769,346.046,-81.554,-177.339,10.904,149.503
C00688=1129.766,346.293,-81.590,-177.337,10.907,149.503
C00689=1129.762,346.542,-81.625,-177.333,10.909,149.502
C00690=1129.757,346.789,-81.659,-177.330,10.912,149.502
C00691=1129.754,347.036,-81.694,-177.327,10.914,149.502
C00692=1129.750,347.284,-81.728,-177.323,10.917,149.502
C00693=1129.746,347.531,-81.764,-177.320,10.919,149.502
C00694=1129.742,347.779,-81.799,-177.317,10.922,149.501
C00695=1129.738,347.992,-81.829,-177.314,10.924,149.501
C00696=1129.735,348.205,-81.859,-177.312,10.925,149.501
C00697=1129.731,348.417,-81.889,-177.308,10.928,149.501
C00698=1129.729,348.630,-81.919,-177.306,10.930,149.501
C00699=1129.726,348.844,-81.950,-177.303,10.932,149.500
C00700=1129.722,349.056,-81.980,-177.301,10.934,149.500
C00701=1129.719,349.269,-82.010,-177.297,10.937,149.500
C00702=1129.715,349.482,-82.040,-177.295,10.938,149.500
C00703=1129.711,349.730,-82.075,-177.291,10.941,149.500
C00704=1129.707,349.977,-82.110,-177.287,10.944,149.499
C00705=1129.703,350.224,-82.146,-177.284,10.947,149.499
C00706=1129.699,350.472,-82.180,-177.280,10.950,149.499
C00707=1129.695,350.720,-82.216,-177.276,10.952,149.499
C00708=1129.692,350.967,-82.251,-177.273,10.954,149.498
C00709=1129.687,351.215,-82.286,-177.269,10.958,149.498
C00710=1129.684,351.462,-82.322,-177.265,10.960,149.498
C00711=1129.680,351.710,-82.357,-177.262,10.962,149.498
C00712=1129.676,351.957,-82.393,-177.258,10.966,149.497
C00713=1129.672,352.205,-82.427,-177.255,10.968,149.497
C00714=1129.668,352.452,-82.463,-177.251,10.970,149.497
C00715=1129.664,352.700,-82.498,-177.247,10.973,149.497
C00716=1129.661,352.947,-82.534,-177.244,10.976,149.496
C00717=1129.656,353.194,-82.569,-177.241,10.978,149.496
C00718=1129.653,353.441,-82.604,-177.236,10.981,149.496
C00719=1129.649,353.690,-82.639,-177.233,10.984,149.495
C00720=1129.645,353.937,-82.675,-177.230,10.986,149.495
C00721=1129.641,354.184,-82.710,-177.226,10.988,149.495
C00722=1129.637,354.431,-82.746,-177.222,10.992,149.495
C00723=1129.634,354.679,-82.781,-177.219,10.994,149.494
C00724=1129.630,354.926,-82.817,-177.215,10.996,149.494
C00725=1129.626,355.174,-82.852,-177.212,10.999,149.494
C00726=1129.623,355.421,-82.888,-177.208,11.002,149.494
C00727=1129.618,355.668,-82.924,-177.204,11.004,149.493
C00728=1129.614,355.916,-82.959,-177.201,11.007,149.493
C00729=1129.610,356.163,-82.995,-177.197,11.009,149.493
C00730=1129.607,356.411,-83.030,-177.194,11.011,149.493
C00731=1129.603,356.658,-83.066,-177.191,11.014,149.492
C00732=1129.599,356.906,-83.101,-177.186,11.017,149.492
C00733=1129.595,357.154,-83.137,-177.183,11.019,149.492
C00734=1129.591,357.401,-83.173,-177.180,11.022,149.492
C00735=1129.587,357.647,-83.209,-177.176,11.024,149.491
C00736=1129.584,357.895,-83.244,-177.173,11.026,149.491
C00737=1129.580,358.142,-83.280,-177.169,11.029,149.491
C00738=1129.576,358.390,-83.316,-177.166,11.031,149.490
C00739=1129.572,358.638,-83.352,-177.163,11.034,149.490
C00740=1129.568,358.885,-83.387,-177.158,11.037,149.490
C00741=1129.565,359.132,-83.423,-177.155,11.039,149.490
C00742=1129.560,359.380,-83.460,-177.152,11.042,149.489
C00743=1129.557,359.627,-83.495,-177.148,11.044,149.489
C00744=1129.553,359.875,-83.531,-177.145,11.046,149.489
C00745=1129.549,360.122,-83.568,-177.142,11.049,149.489
C00746=1129.545,360.369,-83.603,-177.138,11.051,149.488
C00747=1129.541,360.616,-83.638,-177.135,11.053,149.488
C00748=1129.538,360.863,-83.675,-177.131,11.056,149.488
C00749=1129.533,361.111,-83.711,-177.128,11.058,149.488
C00750=1129.530,361.359,-83.746,-177.125,11.061,149.487
C00751=1129.527,361.571,-83.778,-177.122,11.062,149.487
C00752=1129.524,361.784,-83.809,-177.119,11.065,149.487
C00753=1129.520,361.997,-83.839,-177.116,11.066,149.487
C00754=1129.517,362.210,-83.871,-177.113,11.069,149.486
C00755=1129.514,362.422,-83.902,-177.110,11.071,149.486
C00756=1129.510,362.635,-83.932,-177.107,11.072,149.486
C00757=1129.507,362.848,-83.963,-177.104,11.075,149.486
C00758=1129.504,363.060,-83.995,-177.102,11.077,149.486
C00759=1129.500,363.308,-84.031,-177.098,11.079,149.485
C00760=1129.496,363.555,-84.067,-177.095,11.081,149.485
C00761=1129.492,363.803,-84.103,-177.091,11.084,149.485
C00762=1129.489,364.050,-84.139,-177.088,11.086,149.485
C00763=1129.484,364.298,-84.176,-177.085,11.089,149.484
C00764=1129.481,364.544,-84.212,-177.082,11.091,149.484
C00765=1129.477,364.792,-84.247,-177.078,11.093,149.484
C00766=1129.473,365.039,-84.284,-177.075,11.096,149.484
C00767=1129.470,365.286,-84.321,-177.071,11.098,149.483
C00768=1129.465,365.534,-84.357,-177.069,11.100,149.483
C00769=1129.463,365.781,-84.393,-177.065,11.103,149.483
C00770=1129.458,366.029,-84.429,-177.062,11.105,149.483
C00771=1129.455,366.276,-84.466,-177.059,11.107,149.482
C00772=1129.451,366.523,-84.503,-177.055,11.110,149.482
C00773=1129.446,366.771,-84.539,-177.052,11.112,149.482
C00774=1129.443,367.018,-84.575,-177.048,11.115,149.482
C00775=1129.439,367.265,-84.612,-177.046,11.116,149.481
C00776=1129.435,367.513,-84.647,-177.042,11.119,149.481
C00777=1129.431,367.760,-84.684,-177.039,11.121,149.481
C00778=1129.428,368.007,-84.720,-177.036,11.124,149.481
C00779=1129.424,368.254,-84.757,-177.032,11.126,149.481
C00780=1129.420,368.502,-84.794,-177.030,11.128,149.480
C00781=1129.416,368.749,-84.830,-177.026,11.130,149.480
C00782=1129.412,368.997,-84.867,-177.023,11.133,149.480
C00783=1129.409,369.243,-84.903,-177.020,11.135,149.480
C00784=1129.405,369.491,-84.940,-177.017,11.138,149.479
C00785=1129.401,369.738,-84.977,-177.014,11.139,149.479
C00786=1129.397,369.985,-85.013,-177.011,11.142,149.479
C00787=1129.393,370.232,-85.049,-177.007,11.144,149.479
C00788=1129.390,370.480,-85.087,-177.004,11.147,149.479
C00789=1129.386,370.727,-85.123,-177.001,11.149,149.478
C00790=1129.382,370.974,-85.160,-176.998,11.151,149.478
C00791=1129.378,371.222,-85.197,-176.995,11.154,149.478
C00792=1129.375,371.469,-85.233,-176.991,11.156,149.478
C00793=1129.371,371.716,-85.270,-176.989,11.158,149.478
C00794=1129.367,371.964,-85.307,-176.986,11.160,149.477
C00795=1129.363,372.211,-85.344,-176.983,11.163,149.477
C00796=1129.360,372.458,-85.380,-176.979,11.165,149.477
C00797=1129.356,372.705,-85.417,-176.977,11.167,149.477
C00798=1129.352,372.953,-85.454,-176.973,11.170,149.477
C00799=1129.348,373.200,-85.491,-176.970,11.172,149.476
C00800=1129.345,373.447,-85.527,-176.968,11.174,149.476
C00801=1129.341,373.694,-85.564,-176.964,11.177,149.476
C00802=1129.336,373.941,-85.601,-176.961,11.179,149.476
C00803=1129.333,374.189,-85.638,-176.958,11.181,149.476
C00804=1129.330,374.436,-85.674,-176.956,11.184,149.476
C00805=1129.325,374.683,-85.711,-176.952,11.186,149.475
C00806=1129.321,374.930,-85.748,-176.950,11.188,149.475
C00807=1129.319,375.142,-85.780,-176.947,11.190,149.475
C00808=1129.315,375.356,-85.812,-176.944,11.192,149.475
C00809=1129.312,375.569,-85.844,-176.942,11.194,149.475
C00810=1129.309,375.781,-85.876,-176.939,11.196,149.475
C00811=1129.306,375.994,-85.908,-176.937,11.198,149.475
C00812=1129.302,376.206,-85.940,-176.934,11.200,149.474
C00813=1129.299,376.419,-85.971,-176.932,11.202,149.474
C00814=1129.296,376.632,-86.003,-176.930,11.204,149.474
C00815=1129.293,376.878,-86.040,-176.926,11.206,149.474
C00816=1129.288,377.125,-86.077,-176.923,11.209,149.474
C00817=1129.285,377.373,-86.114,-176.921,11.211,149.474
C00818=1129.281,377.620,-86.151,-176.917,11.213,149.473
C00819=1129.277,377.867,-86.189,-176.915,11.215,149.473
C00820=1129.274,378.115,-86.226,-176.912,11.218,149.473
C00821=1129.269,378.362,-86.263,-176.909,11.221,149.473
C00822=1129.266,378.608,-86.300,-176.906,11.222,149.473
C00823=1129.262,378.856,-86.337,-176.903,11.225,149.473
C00824=1129.258,379.104,-86.375,-176.901,11.227,149.473
C00825=1129.254,379.350,-86.412,-176.898,11.230,149.473
C00826=1129.250,379.597,-86.449,-176.895,11.232,149.473
C00827=1129.247,379.845,-86.486,-176.892,11.234,149.472
C00828=1129.243,380.092,-86.524,-176.889,11.237,149.472
C00829=1129.239,380.340,-86.561,-176.887,11.239,149.472
C00830=1129.236,380.586,-86.599,-176.884,11.241,149.472
C00831=1129.232,380.833,-86.635,-176.882,11.243,149.472
C00832=1129.228,381.081,-86.673,-176.878,11.246,149.472
C00833=1129.224,381.328,-86.710,-176.875,11.249,149.472
C00834=1129.220,381.574,-86.748,-176.873,11.251,149.472
C00835=1129.217,381.822,-86.785,-176.870,11.254,149.472
C00836=1129.213,382.069,-86.823,-176.867,11.255,149.472
C00837=1129.210,382.317,-86.860,-176.865,11.258,149.472
C00838=1129.206,382.563,-86.897,-176.862,11.260,149.472
C00839=1129.202,382.811,-86.934,-176.859,11.263,149.472
C00840=1129.199,383.058,-86.972,-176.857,11.265,149.471
C00841=1129.195,383.305,-87.009,-176.854,11.267,149.471
C00842=1129.191,383.552,-87.047,-176.852,11.270,149.471
C00843=1129.188,383.799,-87.085,-176.851,11.271,149.472
C00844=1129.183,384.046,-87.121,-176.849,11.273,149.472
C00845=1129.180,384.294,-87.160,-176.848,11.275,149.472
C00846=1129.175,384.541,-87.197,-176.846,11.277,149.472
C00847=1129.172,384.788,-87.235,-176.845,11.278,149.472
C00848=1129.168,385.035,-87.272,-176.844,11.280,149.472
C00849=1129.165,385.283,-87.310,-176.843,11.282,149.472
C00850=1129.161,385.529,-87.347,-176.841,11.284,149.472
C00851=1129.158,385.776,-87.385,-176.839,11.286,149.472
C00852=1129.154,386.024,-87.422,-176.839,11.287,149.473
C00853=1129.150,386.270,-87.459,-176.837,11.289,149.473
C00854=1129.146,386.518,-87.498,-176.835,11.291,149.473
C00855=1129.142,386.765,-87.535,-176.835,11.293,149.473
C00856=1129.139,387.012,-87.573,-176.833,11.295,149.473
C00857=1129.135,387.259,-87.610,-176.832,11.296,149.473
C00858=1129.132,387.507,-87.648,-176.831,11.299,149.474
C00859=1129.128,387.753,-87.685,-176.830,11.301,149.474
C00860=1129.125,388.000,-87.723,-176.829,11.303,149.474
C00861=1129.120,388.247,-87.761,-176.828,11.304,149.474
C00862=1129.117,388.495,-87.798,-176.826,11.307,149.474
C00863=1129.113,388.708,-87.831,-176.825,11.309,149.475
C00864=1129.110,388.920,-87.863,-176.824,11.311,149.475
C00865=1129.107,389.132,-87.896,-176.823,11.312,149.475
C00866=1129.103,389.344,-87.928,-176.822,11.314,149.475
C00867=1129.101,389.557,-87.961,-176.821,11.316,149.476
C00868=1129.098,389.769,-87.993,-176.820,11.318,149.476
C00869=1129.094,389.982,-88.025,-176.819,11.320,149.476
C00870=1129.091,390.195,-88.058,-176.818,11.321,149.476
C00871=1129.087,390.442,-88.096,-176.817,11.323,149.476
C00872=1129.084,390.689,-88.133,-176.817,11.326,149.477
C00873=1129.080,390.936,-88.171,-176.815,11.328,149.477
C00874=1129.077,391.182,-88.209,-176.815,11.330,149.478
C00875=1129.072,391.431,-88.246,-176.814,11.332,149.478
C00876=1129.069,391.677,-88.284,-176.812,11.335,149.478
C00877=1129.065,391.924,-88.322,-176.812,11.337,149.479
C00878=1129.062,392.171,-88.360,-176.811,11.339,149.479
C00879=1129.058,392.418,-88.398,-176.810,11.342,149.479
C00880=1129.054,392.665,-88.436,-176.809,11.344,149.480
C00881=1129.051,392.912,-88.474,-176.808,11.346,149.480
C00882=1129.047,393.160,-88.510,-176.807,11.349,149.480
C00883=1129.043,393.407,-88.548,-176.807,11.351,149.481
C00884=1129.039,393.654,-88.587,-176.806,11.353,149.481
C00885=1129.036,393.901,-88.625,-176.805,11.356,149.482
C00886=1129.032,394.148,-88.662,-176.804,11.358,149.482
C00887=1129.028,394.395,-88.701,-176.803,11.361,149.483
C00888=1129.025,394.642,-88.739,-176.803,11.363,149.483
C00889=1129.021,394.889,-88.776,-176.802,11.365,149.484
C00890=1129.018,395.136,-88.814,-176.801,11.369,149.484
C00891=1129.013,395.383,-88.852,-176.801,11.371,149.484
C00892=1129.010,395.631,-88.889,-176.799,11.374,149.485
C00893=1129.006,395.878,-88.927,-176.799,11.376,149.485
C00894=1129.002,396.125,-88.966,-176.798,11.379,149.486
C00895=1128.998,396.372,-89.003,-176.798,11.382,149.487
C00896=1128.995,396.619,-89.041,-176.797,11.384,149.487
C00897=1128.991,396.866,-89.079,-176.797,11.387,149.488
C00898=1128.987,397.113,-89.117,-176.796,11.389,149.488
C00899=1128.984,397.360,-89.155,-176.795,11.392,149.489
C00900=1128.980,397.607,-89.193,-176.795,11.395,149.489
C00901=1128.977,397.855,-89.231,-176.794,11.398,149.490
C00902=1128.973,398.101,-89.269,-176.794,11.400,149.491
C00903=1128.969,398.349,-89.307,-176.793,11.404,149.491
C00904=1128.965,398.595,-89.345,-176.793,11.406,149.492
C00905=1128.962,398.843,-89.383,-176.792,11.410,149.493
C00906=1128.958,399.090,-89.421,-176.792,11.412,149.493
C00907=1128.954,399.337,-89.459,-176.791,11.415,149.494
C00908=1128.951,399.584,-89.497,-176.791,11.418,149.494
C00909=1128.946,399.831,-89.535,-176.791,11.422,149.495
C00910=1128.944,400.078,-89.574,-176.790,11.425,149.496
C00911=1128.940,400.324,-89.611,-176.790,11.427,149.497
C00912=1128.936,400.572,-89.650,-176.789,11.431,149.497
C00913=1128.933,400.819,-89.688,-176.789,11.433,149.498
C00914=1128.928,401.066,-89.726,-176.789,11.437,149.499
C00915=1128.925,401.313,-89.764,-176.789,11.440,149.499
C00916=1128.921,401.560,-89.801,-176.789,11.443,149.500
C00917=1128.917,401.807,-89.840,-176.788,11.447,149.501
C00918=1128.914,402.055,-89.878,-176.788,11.449,149.502
C00919=1128.911,402.267,-89.911,-176.788,11.452,149.502
C00920=1128.907,402.479,-89.944,-176.787,11.455,149.503
C00921=1128.904,402.691,-89.976,-176.787,11.458,149.504
C00922=1128.901,402.904,-90.009,-176.788,11.461,149.505
C00923=1128.898,403.116,-90.042,-176.787,11.464,149.505
C00924=1128.894,403.328,-90.075,-176.787,11.467,149.506
C00925=1128.892,403.541,-90.108,-176.787,11.470,149.507
C00926=1128.889,403.753,-90.140,-176.787,11.472,149.507
C00927=1128.885,404.001,-90.179,-176.787,11.476,149.508
C00928=1128.881,404.247,-90.216,-176.787,11.480,149.509
C00929=1128.877,404.494,-90.256,-176.787,11.483,149.510
C00930=1128.874,404.741,-90.293,-176.787,11.486,149.511
C00931=1128.870,404.988,-90.331,-176.787,11.490,149.512
C00932=1128.867,405.236,-90.370,-176.787,11.494,149.513
C00933=1128.863,405.482,-90.407,-176.787,11.497,149.514
C00934=1128.859,405.729,-90.446,-176.787,11.501,149.515
C00935=1128.856,405.976,-90.484,-176.787,11.505,149.516
C00936=1128.851,406.223,-90.523,-176.787,11.509,149.517
C00937=1128.848,406.471,-90.561,-176.788,11.512,149.518
C00938=1128.845,406.718,-90.600,-176.788,11.516,149.519
C00939=1128.841,406.964,-90.637,-176.787,11.519,149.520
C00940=1128.837,407.212,-90.676,-176.787,11.523,149.521
C00941=1128.834,407.459,-90.714,-176.788,11.527,149.522
C00942=1128.830,407.705,-90.752,-176.789,11.531,149.523
C00943=1128.826,407.953,-90.791,-176.789,11.535,149.524
C00944=1128.823,408.200,-90.829,-176.789,11.539,149.525
C00945=1128.819,408.447,-90.867,-176.789,11.543,149.526
C00946=1128.816,408.693,-90.905,-176.789,11.547,149.527
C00947=1128.812,408.941,-90.944,-176.789,11.551,149.529
C00948=1128.808,409.188,-90.982,-176.790,11.554,149.530
C00949=1128.804,409.434,-91.021,-176.790,11.559,149.531
C00950=1128.801,409.682,-91.059,-176.791,11.563,149.532
C00951=1128.797,409.929,-91.097,-176.791,11.567,149.533
C00952=1128.793,410.176,-91.135,-176.791,11.571,149.534
C00953=1128.790,410.423,-91.174,-176.792,11.576,149.536
C00954=1128.785,410.670,-91.212,-176.792,11.580,149.537
C00955=1128.782,410.917,-91.250,-176.793,11.584,149.538
C00956=1128.779,411.164,-91.289,-176.793,11.589,149.539
C00957=1128.775,411.411,-91.327,-176.794,11.593,149.541
C00958=1128.771,411.657,-91.366,-176.794,11.597,149.542
C00959=1128.768,411.905,-91.404,-176.795,11.602,149.543
C00960=1128.764,412.152,-91.443,-176.796,11.606,149.544
C00961=1128.761,412.398,-91.481,-176.796,11.611,149.546
C00962=1128.757,412.646,-91.520,-176.797,11.615,149.547
C00963=1128.753,412.893,-91.557,-176.797,11.620,149.548
C00964=1128.749,413.139,-91.596,-176.798,11.624,149.550
C00965=1128.745,413.387,-91.635,-176.799,11.629,149.551
C00966=1128.742,413.634,-91.674,-176.799,11.633,149.552
C00967=1128.738,413.881,-91.712,-176.800,11.638,149.554
C00968=1128.735,414.128,-91.750,-176.801,11.643,149.555
C00969=1128.732,414.374,-91.788,-176.802,11.647,149.557
C00970=1128.730,414.622,-91.827,-176.803,11.652,149.558
C00971=1128.728,414.869,-91.865,-176.804,11.656,149.560
C00972=1128.727,415.116,-91.903,-176.804,11.661,149.561
C00973=1128.726,415.363,-91.941,-176.806,11.666,149.563
C00974=1128.726,415.610,-91.979,-176.806,11.672,149.564
C00975=1128.726,415.822,-92.012,-176.807,11.675,149.565
C00976=1128.727,416.035,-92.044,-176.808,11.680,149.567
C00977=1128.729,416.247,-92.077,-176.809,11.684,149.568
C00978=1128.731,416.459,-92.109,-176.810,11.688,149.569
C00979=1128.733,416.671,-92.141,-176.810,11.693,149.571
C00980=1128.735,416.883,-92.174,-176.812,11.696,149.572
C00981=1128.739,417.096,-92.205,-176.813,11.701,149.573
C00982=1128.742,417.308,-92.238,-176.814,11.706,149.575
C00983=1128.324,417.307,-92.301,-176.806,11.710,149.574
C00984=1128.320,417.095,-92.269,-176.805,11.705,149.573
C00985=1128.316,416.883,-92.237,-176.804,11.701,149.571
C00986=1128.314,416.671,-92.204,-176.803,11.697,149.570
C00987=1128.311,416.459,-92.172,-176.803,11.693,149.569
C00988=1128.310,416.246,-92.140,-176.802,11.688,149.567
C00989=1128.308,416.035,-92.107,-176.801,11.684,149.566
C00990=1128.307,415.822,-92.075,-176.800,11.680,149.565
C00991=1128.307,415.610,-92.042,-176.799,11.675,149.563
C00992=1128.307,415.363,-92.003,-176.798,11.670,149.562
C00993=1128.308,415.116,-91.966,-176.797,11.666,149.560
C00994=1128.308,414.869,-91.927,-176.797,11.661,149.559
C00995=1128.310,414.622,-91.889,-176.796,11.656,149.558
C00996=1128.313,414.374,-91.851,-176.795,11.652,149.556
C00997=1128.316,414.128,-91.812,-176.795,11.646,149.555
C00998=1128.319,413.881,-91.774,-176.794,11.642,149.553
C00999=1128.323,413.634,-91.735,-176.793,11.637,149.552
C01000=1128.326,413.387,-91.698,-176.792,11.632,149.550
C01001=1128.330,413.140,-91.658,-176.792,11.628,149.549
C01002=1128.334,412.892,-91.620,-176.791,11.623,149.548
C01003=1128.337,412.645,-91.582,-176.790,11.619,149.547
C01004=1128.341,412.399,-91.543,-176.790,11.614,149.545
C01005=1128.344,412.152,-91.505,-176.789,11.610,149.544
C01006=1128.348,411.905,-91.466,-176.789,11.605,149.542
C01007=1128.352,411.658,-91.428,-176.788,11.600,149.541
C01008=1128.356,411.411,-91.390,-176.788,11.596,149.540
C01009=1128.359,411.164,-91.350,-176.788,11.592,149.539
C01010=1128.363,410.916,-91.313,-176.787,11.587,149.537
C01011=1128.367,410.670,-91.274,-176.787,11.583,149.536
C01012=1128.370,410.423,-91.236,-176.786,11.579,149.535
C01013=1128.374,410.175,-91.197,-176.786,11.574,149.534
C01014=1128.377,409.929,-91.159,-176.786,11.570,149.533
C01015=1128.381,409.682,-91.120,-176.785,11.566,149.531
C01016=1128.385,409.434,-91.082,-176.785,11.562,149.530
C01017=1128.389,409.188,-91.044,-176.785,11.558,149.529
C01018=1128.392,408.941,-91.006,-176.784,11.555,149.528
C01019=1128.396,408.693,-90.967,-176.784,11.550,149.527
C01020=1128.399,408.447,-90.929,-176.783,11.546,149.526
C01021=1128.403,408.200,-90.890,-176.783,11.542,149.525
C01022=1128.406,407.952,-90.852,-176.783,11.538,149.524
C01023=1128.410,407.705,-90.814,-176.783,11.534,149.522
C01024=1128.414,407.459,-90.775,-176.783,11.530,149.521
C01025=1128.418,407.211,-90.737,-176.783,11.526,149.520
C01026=1128.421,406.964,-90.699,-176.783,11.522,149.519
C01027=1128.425,406.718,-90.660,-176.782,11.519,149.518
C01028=1128.428,406.471,-90.622,-176.782,11.515,149.517
C01029=1128.432,406.223,-90.584,-176.782,11.511,149.516
C01030=1128.436,405.976,-90.546,-176.782,11.507,149.515
C01031=1128.440,405.729,-90.507,-176.782,11.503,149.514
C01032=1128.443,405.482,-90.469,-176.782,11.500,149.513
C01033=1128.447,405.235,-90.431,-176.782,11.497,149.513
C01034=1128.451,404.988,-90.393,-176.782,11.493,149.512
C01035=1128.454,404.741,-90.355,-176.782,11.489,149.511
C01036=1128.458,404.494,-90.316,-176.783,11.485,149.510
C01037=1128.461,404.247,-90.278,-176.782,11.482,149.509
C01038=1128.466,404.000,-90.240,-176.783,11.479,149.508
C01039=1128.469,403.753,-90.202,-176.783,11.475,149.507
C01040=1128.472,403.541,-90.169,-176.783,11.472,149.506
C01041=1128.475,403.328,-90.136,-176.783,11.470,149.506
C01042=1128.478,403.116,-90.103,-176.783,11.466,149.505
C01043=1128.482,402.904,-90.070,-176.783,11.463,149.504
C01044=1128.485,402.692,-90.037,-176.783,11.461,149.503
C01045=1128.488,402.479,-90.004,-176.784,11.457,149.503
C01046=1128.491,402.267,-89.972,-176.784,11.455,149.502
C01047=1128.494,402.054,-89.940,-176.784,11.452,149.501
C01048=1128.498,401.807,-89.901,-176.784,11.449,149.501
C01049=1128.502,401.561,-89.863,-176.785,11.445,149.500
C01050=1128.505,401.314,-89.825,-176.785,11.442,149.499
C01051=1128.509,401.066,-89.786,-176.785,11.439,149.498
C01052=1128.512,400.820,-89.749,-176.786,11.435,149.498
C01053=1128.516,400.572,-89.710,-176.786,11.433,149.497
C01054=1128.520,400.325,-89.673,-176.786,11.430,149.496
C01055=1128.523,400.078,-89.635,-176.786,11.427,149.496
C01056=1128.527,399.831,-89.596,-176.787,11.424,149.495
C01057=1128.531,399.584,-89.559,-176.788,11.420,149.494
C01058=1128.535,399.336,-89.520,-176.788,11.418,149.494
C01059=1128.539,399.090,-89.482,-176.789,11.414,149.493
C01060=1128.542,398.843,-89.445,-176.789,11.412,149.492
C01061=1128.546,398.595,-89.406,-176.789,11.409,149.491
C01062=1128.549,398.349,-89.368,-176.790,11.406,149.491
C01063=1128.553,398.102,-89.330,-176.791,11.403,149.490
C01064=1128.557,397.855,-89.292,-176.791,11.400,149.490
C01065=1128.560,397.608,-89.254,-176.791,11.397,149.489
C01066=1128.564,397.361,-89.216,-176.792,11.394,149.488
C01067=1128.568,397.113,-89.178,-176.793,11.392,149.488
C01068=1128.571,396.866,-89.140,-176.794,11.388,149.487
C01069=1128.575,396.620,-89.102,-176.794,11.386,149.487
C01070=1128.579,396.372,-89.064,-176.795,11.383,149.486
C01071=1128.583,396.125,-89.026,-176.795,11.381,149.486
C01072=1128.586,395.878,-88.989,-176.796,11.378,149.485
C01073=1128.591,395.631,-88.951,-176.797,11.375,149.485
C01074=1128.594,395.383,-88.913,-176.798,11.372,149.484
C01075=1128.598,395.137,-88.875,-176.798,11.370,149.484
C01076=1128.602,394.889,-88.837,-176.799,11.367,149.483
C01077=1128.605,394.643,-88.799,-176.800,11.365,149.483
C01078=1128.609,394.395,-88.761,-176.800,11.363,149.482
C01079=1128.612,394.148,-88.723,-176.801,11.360,149.482
C01080=1128.616,393.901,-88.685,-176.802,11.357,149.481
C01081=1128.620,393.654,-88.647,-176.803,11.355,149.481
C01082=1128.623,393.407,-88.609,-176.804,11.353,149.481
C01083=1128.627,393.160,-88.571,-176.805,11.350,149.480
C01084=1128.631,392.913,-88.533,-176.806,11.348,149.480
C01085=1128.635,392.665,-88.496,-176.806,11.345,149.479
C01086=1128.638,392.419,-88.458,-176.808,11.343,149.479
C01087=1128.642,392.171,-88.420,-176.808,11.341,149.479
C01088=1128.646,391.925,-88.382,-176.810,11.338,149.478
C01089=1128.649,391.677,-88.344,-176.811,11.336,149.478
C01090=1128.653,391.431,-88.307,-176.811,11.334,149.478
C01091=1128.656,391.183,-88.270,-176.812,11.331,149.477
C01092=1128.661,390.936,-88.231,-176.813,11.329,149.477
C01093=1128.664,390.689,-88.194,-176.815,11.326,149.477
C01094=1128.668,390.442,-88.156,-176.816,11.325,149.476
C01095=1128.671,390.195,-88.118,-176.817,11.323,149.476
C01096=1128.675,389.983,-88.085,-176.817,11.321,149.476
C01097=1128.678,389.770,-88.053,-176.818,11.319,149.476
C01098=1128.681,389.558,-88.021,-176.819,11.317,149.475
C01099=1128.684,389.345,-87.989,-176.820,11.315,149.475
C01100=1128.688,389.132,-87.956,-176.821,11.313,149.475
C01101=1128.691,388.920,-87.923,-176.822,11.312,149.475
C01102=1128.694,388.708,-87.891,-176.823,11.310,149.475
C01103=1128.697,388.495,-87.859,-176.824,11.308,149.474
C01104=1128.700,388.248,-87.821,-176.826,11.305,149.474
C01105=1128.704,388.001,-87.784,-176.827,11.304,149.474
C01106=1128.708,387.754,-87.746,-176.828,11.302,149.474
C01107=1128.712,387.507,-87.708,-176.830,11.300,149.473
C01108=1128.715,387.260,-87.670,-176.830,11.298,149.473
C01109=1128.719,387.012,-87.633,-176.832,11.296,149.473
C01110=1128.723,386.765,-87.595,-176.833,11.293,149.473
C01111=1128.726,386.519,-87.558,-176.834,11.292,149.473
C01112=1128.730,386.271,-87.520,-176.836,11.290,149.473
C01113=1128.734,386.024,-87.483,-176.837,11.288,149.472
C01114=1128.738,385.777,-87.445,-176.838,11.286,149.472
C01115=1128.742,385.529,-87.407,-176.840,11.284,149.472
C01116=1128.746,385.283,-87.370,-176.841,11.283,149.472
C01117=1128.749,385.035,-87.332,-176.843,11.280,149.472
C01118=1128.753,384.788,-87.295,-176.844,11.279,149.472
C01119=1128.756,384.541,-87.257,-176.845,11.277,149.472
C01120=1128.760,384.294,-87.220,-176.847,11.276,149.472
C01121=1128.763,384.047,-87.182,-176.848,11.273,149.471
C01122=1128.767,383.800,-87.145,-176.850,11.272,149.471
C01123=1128.772,383.552,-87.107,-176.851,11.270,149.471
C01124=1128.775,383.305,-87.069,-176.853,11.268,149.471
C01125=1128.779,383.059,-87.032,-176.856,11.265,149.471
C01126=1128.782,382.811,-86.995,-176.858,11.263,149.471
C01127=1128.786,382.564,-86.957,-176.861,11.261,149.471
C01128=1128.790,382.317,-86.920,-176.864,11.259,149.471
C01129=1128.793,382.070,-86.882,-176.867,11.256,149.472
C01130=1128.798,381.823,-86.845,-176.869,11.254,149.472
C01131=1128.801,381.575,-86.807,-176.872,11.251,149.472
C01132=1128.805,381.328,-86.771,-176.874,11.249,149.472
C01133=1128.809,381.081,-86.733,-176.878,11.247,149.472
C01134=1128.812,380.834,-86.696,-176.880,11.244,149.472
C01135=1128.816,380.587,-86.658,-176.883,11.242,149.472
C01136=1128.820,380.340,-86.621,-176.886,11.239,149.472
C01137=1128.823,380.093,-86.583,-176.888,11.237,149.472
C01138=1128.827,379.845,-86.547,-176.891,11.235,149.472
C01139=1128.831,379.597,-86.509,-176.894,11.233,149.473
C01140=1128.835,379.351,-86.472,-176.897,11.230,149.473
C01141=1128.839,379.104,-86.435,-176.900,11.228,149.473
C01142=1128.842,378.856,-86.397,-176.902,11.226,149.473
C01143=1128.846,378.609,-86.360,-176.906,11.223,149.473
C01144=1128.850,378.362,-86.323,-176.908,11.221,149.473
C01145=1128.853,378.115,-86.285,-176.911,11.219,149.473
C01146=1128.857,377.868,-86.248,-176.914,11.216,149.473
C01147=1128.861,377.620,-86.212,-176.917,11.214,149.474
C01148=1128.866,377.373,-86.175,-176.920,11.211,149.474
C01149=1128.868,377.126,-86.137,-176.923,11.209,149.474
C01150=1128.872,376.879,-86.100,-176.925,11.207,149.474
C01151=1128.876,376.632,-86.064,-176.929,11.204,149.474
C01152=1128.880,376.420,-86.031,-176.931,11.202,149.474
C01153=1128.883,376.207,-86.000,-176.933,11.201,149.474
C01154=1128.886,375.994,-85.968,-176.936,11.198,149.474
C01155=1128.889,375.782,-85.936,-176.938,11.197,149.475
C01156=1128.892,375.569,-85.905,-176.941,11.195,149.475
C01157=1128.896,375.357,-85.872,-176.944,11.192,149.475
C01158=1128.899,375.144,-85.841,-176.946,11.190,149.475
C01159=1128.903,374.931,-85.809,-176.949,11.189,149.475
C01160=1128.906,374.683,-85.772,-176.952,11.186,149.475
C01161=1128.909,374.437,-85.735,-176.955,11.184,149.475
C01162=1128.913,374.190,-85.698,-176.958,11.182,149.476
C01163=1128.917,373.943,-85.661,-176.961,11.179,149.476
C01164=1128.921,373.695,-85.624,-176.963,11.177,149.476
C01165=1128.924,373.448,-85.587,-176.967,11.175,149.476
C01166=1128.928,373.201,-85.551,-176.970,11.172,149.476
C01167=1128.932,372.954,-85.514,-176.973,11.170,149.477
C01168=1128.936,372.706,-85.477,-176.976,11.168,149.477
C01169=1128.939,372.459,-85.440,-176.979,11.165,149.477
C01170=1128.943,372.212,-85.403,-176.982,11.163,149.477
C01171=1128.947,371.964,-85.367,-176.985,11.161,149.477
C01172=1128.951,371.717,-85.330,-176.988,11.158,149.477
C01173=1128.954,371.470,-85.293,-176.991,11.156,149.478
C01174=1128.958,371.222,-85.256,-176.994,11.154,149.478
C01175=1128.962,370.975,-85.219,-176.997,11.152,149.478
C01176=1128.966,370.728,-85.183,-177.001,11.149,149.478
C01177=1128.970,370.481,-85.146,-177.004,11.147,149.479
C01178=1128.974,370.233,-85.110,-177.007,11.145,149.479
C01179=1128.977,369.986,-85.073,-177.010,11.143,149.479
C01180=1128.981,369.739,-85.037,-177.013,11.140,149.479
C01181=1128.985,369.491,-85.000,-177.017,11.138,149.479
C01182=1128.989,369.245,-84.963,-177.020,11.135,149.480
C01183=1128.993,368.997,-84.927,-177.023,11.134,149.480
C01184=1128.997,368.750,-84.890,-177.026,11.131,149.480
C01185=1129.000,368.503,-84.854,-177.029,11.129,149.480
C01186=1129.004,368.255,-84.817,-177.032,11.126,149.481
C01187=1129.007,368.008,-84.781,-177.036,11.124,149.481
C01188=1129.011,367.761,-84.744,-177.038,11.122,149.481
C01189=1129.016,367.513,-84.708,-177.042,11.120,149.481
C01190=1129.019,367.266,-84.671,-177.045,11.117,149.481
C01191=1129.023,367.019,-84.635,-177.048,11.115,149.482
C01192=1129.027,366.771,-84.599,-177.052,11.112,149.482
C01193=1129.031,366.524,-84.562,-177.055,11.110,149.482
C01194=1129.034,366.277,-84.526,-177.058,11.108,149.482
C01195=1129.039,366.029,-84.490,-177.061,11.105,149.482
C01196=1129.042,365.783,-84.454,-177.064,11.103,149.483
C01197=1129.046,365.535,-84.416,-177.068,11.101,149.483
C01198=1129.049,365.287,-84.381,-177.071,11.098,149.483
C01199=1129.053,365.040,-84.344,-177.075,11.096,149.484
C01200=1129.057,364.792,-84.308,-177.078,11.093,149.484
C01201=1129.061,364.545,-84.271,-177.081,11.091,149.484
C01202=1129.064,364.298,-84.235,-177.084,11.088,149.484
C01203=1129.069,364.051,-84.199,-177.087,11.087,149.484
C01204=1129.072,363.804,-84.163,-177.091,11.085,149.485
C01205=1129.077,363.556,-84.127,-177.094,11.082,149.485
C01206=1129.080,363.309,-84.090,-177.097,11.080,149.485
C01207=1129.084,363.062,-84.055,-177.101,11.077,149.485
C01208=1129.087,362.849,-84.024,-177.104,11.075,149.486
C01209=1129.090,362.636,-83.993,-177.107,11.073,149.486
C01210=1129.094,362.423,-83.962,-177.109,11.071,149.486
C01211=1129.097,362.211,-83.930,-177.113,11.069,149.486
C01212=1129.100,361.998,-83.899,-177.115,11.067,149.487
C01213=1129.104,361.785,-83.868,-177.119,11.065,149.487
C01214=1129.107,361.572,-83.837,-177.121,11.063,149.487
C01215=1129.110,361.359,-83.806,-177.124,11.060,149.487
C01216=1129.114,361.113,-83.771,-177.128,11.058,149.488
C01217=1129.118,360.865,-83.735,-177.131,11.056,149.488
C01218=1129.122,360.618,-83.698,-177.135,11.053,149.488
C01219=1129.126,360.370,-83.663,-177.138,11.051,149.488
C01220=1129.129,360.123,-83.627,-177.142,11.049,149.489
C01221=1129.133,359.876,-83.590,-177.145,11.046,149.489
C01222=1129.137,359.628,-83.555,-177.148,11.044,149.489
C01223=1129.141,359.381,-83.519,-177.151,11.041,149.489
C01224=1129.144,359.133,-83.484,-177.155,11.039,149.490
C01225=1129.148,358.886,-83.447,-177.158,11.037,149.490
C01226=1129.152,358.639,-83.411,-177.162,11.034,149.490
C01227=1129.156,358.391,-83.376,-177.165,11.032,149.490
C01228=1129.159,358.144,-83.340,-177.169,11.030,149.491
C01229=1129.164,357.896,-83.304,-177.172,11.027,149.491
C01230=1129.168,357.648,-83.268,-177.175,11.025,149.491
C01231=1129.171,357.402,-83.233,-177.179,11.021,149.491
C01232=1129.175,357.155,-83.197,-177.183,11.019,149.492
C01233=1129.179,356.907,-83.161,-177.186,11.017,149.492
C01234=1129.183,356.659,-83.125,-177.190,11.014,149.492
C01235=1129.187,356.412,-83.090,-177.193,11.012,149.493
C01236=1129.191,356.164,-83.054,-177.197,11.010,149.493
C01237=1129.194,355.917,-83.019,-177.200,11.007,149.493
C01238=1129.198,355.670,-82.984,-177.204,11.004,149.493
C01239=1129.202,355.422,-82.948,-177.208,11.002,149.494
C01240=1129.206,355.175,-82.912,-177.211,10.999,149.494
C01241=1129.210,354.927,-82.876,-177.214,10.997,149.494
C01242=1129.214,354.680,-82.841,-177.218,10.994,149.494
C01243=1129.217,354.432,-82.805,-177.222,10.992,149.495
C01244=1129.222,354.185,-82.770,-177.225,10.989,149.495
C01245=1129.225,353.938,-82.734,-177.229,10.987,149.495
C01246=1129.229,353.690,-82.699,-177.232,10.984,149.496
C01247=1129.233,353.442,-82.664,-177.236,10.981,149.496
C01248=1129.237,353.195,-82.629,-177.239,10.979,149.496
C01249=1129.241,352.948,-82.593,-177.243,10.976,149.496
C01250=1129.245,352.700,-82.558,-177.247,10.973,149.497
C01251=1129.248,352.453,-82.522,-177.250,10.971,149.497
C01252=1129.252,352.205,-82.487,-177.254,10.968,149.497
C01253=1129.257,351.958,-82.452,-177.258,10.965,149.497
C01254=1129.260,351.711,-82.417,-177.261,10.963,149.498
C01255=1129.264,351.463,-82.381,-177.265,10.961,149.498
C01256=1129.268,351.216,-82.346,-177.269,10.957,149.498
C01257=1129.272,350.968,-82.311,-177.272,10.955,149.498
C01258=1129.276,350.721,-82.276,-177.276,10.953,149.499
C01259=1129.279,350.473,-82.240,-177.280,10.950,149.499
C01260=1129.284,350.226,-82.206,-177.283,10.947,149.499
C01261=1129.288,349.978,-82.170,-177.286,10.945,149.499
C01262=1129.291,349.731,-82.134,-177.291,10.942,149.500
C01263=1129.295,349.483,-82.100,-177.294,10.939,149.500
C01264=1129.298,349.270,-82.070,-177.297,10.936,149.500
C01265=1129.302,349.057,-82.039,-177.299,10.935,149.500
C01266=1129.306,348.844,-82.009,-177.303,10.932,149.500
C01267=1129.308,348.631,-81.979,-177.305,10.930,149.501
C01268=1129.312,348.419,-81.949,-177.308,10.929,149.501
C01269=1129.316,348.206,-81.919,-177.311,10.926,149.501
C01270=1129.318,347.993,-81.889,-177.313,10.924,149.501
C01271=1129.322,347.780,-81.858,-177.317,10.922,149.501
C01272=1129.326,347.532,-81.824,-177.320,10.919,149.502
C01273=1129.330,347.286,-81.789,-177.323,10.917,149.502
C01274=1129.334,347.037,-81.754,-177.326,10.915,149.502
C01275=1129.337,346.790,-81.719,-177.329,10.912,149.502
C01276=1129.342,346.542,-81.684,-177.332,10.910,149.502
C01277=1129.346,346.295,-81.649,-177.336,10.907,149.503
C01278=1129.350,346.048,-81.614,-177.339,10.905,149.503
C01279=1129.353,345.800,-81.580,-177.342,10.902,149.503
C01280=1129.357,345.552,-81.544,-177.345,10.900,149.503
C01281=1129.362,345.305,-81.510,-177.348,10.897,149.503
C01282=1129.365,345.057,-81.474,-177.352,10.895,149.503
C01283=1129.369,344.810,-81.440,-177.355,10.892,149.504
C01284=1129.373,344.562,-81.406,-177.358,10.890,149.504
C01285=1129.377,344.314,-81.371,-177.362,10.887,149.504
C01286=1129.381,344.067,-81.336,-177.365,10.885,149.504
C01287=1129.385,343.819,-81.301,-177.368,10.882,149.504
C01288=1129.389,343.572,-81.267,-177.371,10.880,149.505
C01289=1129.393,343.324,-81.231,-177.375,10.877,149.505
C01290=1129.397,343.077,-81.197,-177.378,10.875,149.505
C01291=1129.401,342.829,-81.163,-177.381,10.872,149.505
C01292=1129.405,342.582,-81.128,-177.384,10.870,149.506
C01293=1129.408,342.334,-81.094,-177.387,10.867,149.506
C01294=1129.413,342.087,-81.059,-177.391,10.865,149.506
C01295=1129.417,341.839,-81.024,-177.394,10.862,149.506
C01296=1129.421,341.592,-80.990,-177.397,10.860,149.506
C01297=1129.424,341.344,-80.955,-177.401,10.857,149.507
C01298=1129.429,341.096,-80.921,-177.404,10.855,149.507
C01299=1129.432,340.849,-80.887,-177.407,10.852,149.507
C01300=1129.437,340.601,-80.852,-177.410,10.850,149.507
C01301=1129.440,340.353,-80.818,-177.413,10.848,149.507
C01302=1129.444,340.107,-80.783,-177.416,10.845,149.508
C01303=1129.448,339.858,-80.748,-177.420,10.843,149.508
C01304=1129.452,339.611,-80.714,-177.422,10.840,149.508
C01305=1129.456,339.363,-80.679,-177.426,10.838,149.508
C01306=1129.460,339.116,-80.645,-177.429,10.835,149.508
C01307=1129.464,338.868,-80.610,-177.432,10.833,149.509
C01308=1129.468,338.621,-80.577,-177.436,10.830,149.509
C01309=1129.472,338.373,-80.542,-177.439,10.828,149.509
C01310=1129.476,338.126,-80.508,-177.442,10.825,149.509
C01311=1129.480,337.878,-80.474,-177.445,10.823,149.509
C01312=1129.484,337.630,-80.440,-177.449,10.820,149.510
C01313=1129.488,337.382,-80.405,-177.452,10.818,149.510
C01314=1129.491,337.135,-80.371,-177.455,10.815,149.510
C01315=1129.496,336.887,-80.337,-177.458,10.813,149.510
C01316=1129.500,336.640,-80.303,-177.461,10.810,149.510
C01317=1129.504,336.392,-80.268,-177.465,10.808,149.511
C01318=1129.508,336.145,-80.234,-177.468,10.805,149.511
C01319=1129.512,335.896,-80.200,-177.471,10.802,149.511
C01320=1129.515,335.684,-80.170,-177.474,10.801,149.511
C01321=1129.519,335.471,-80.141,-177.477,10.798,149.511
C01322=1129.522,335.257,-80.112,-177.479,10.796,149.512
C01323=1129.525,335.044,-80.083,-177.482,10.794,149.512
C01324=1129.529,334.832,-80.053,-177.485,10.792,149.512
C01325=1129.532,334.618,-80.024,-177.487,10.790,149.512
C01326=1129.536,334.405,-79.995,-177.491,10.787,149.512
C01327=1129.539,334.193,-79.966,-177.493,10.785,149.512
C01328=1129.543,333.944,-79.931,-177.496,10.783,149.513
C01329=1129.547,333.697,-79.897,-177.499,10.781,149.513
C01330=1129.551,333.450,-79.864,-177.503,10.778,149.513
C01331=1129.555,333.201,-79.829,-177.506,10.775,149.513
C01332=1129.559,332.954,-79.796,-177.509,10.773,149.513
C01333=1129.563,332.707,-79.762,-177.512,10.770,149.514
C01334=1129.566,332.459,-79.728,-177.516,10.768,149.514
C01335=1129.571,332.211,-79.694,-177.519,10.765,149.514
C01336=1129.575,331.964,-79.661,-177.522,10.763,149.514
C01337=1129.578,331.716,-79.626,-177.525,10.760,149.514
C01338=1129.583,331.468,-79.593,-177.529,10.758,149.515
C01339=1129.587,331.221,-79.559,-177.531,10.756,149.515
C01340=1129.591,330.973,-79.526,-177.534,10.753,149.515
C01341=1129.594,330.725,-79.491,-177.537,10.751,149.515
C01342=1129.599,330.477,-79.458,-177.541,10.748,149.515
C01343=1129.603,330.230,-79.424,-177.544,10.746,149.515
C01344=1129.606,329.982,-79.390,-177.547,10.743,149.516
C01345=1129.610,329.734,-79.356,-177.550,10.741,149.516
C01346=1129.614,329.487,-79.323,-177.553,10.738,149.516
C01347=1129.619,329.239,-79.289,-177.557,10.736,149.516
C01348=1129.622,328.991,-79.255,-177.560,10.733,149.516
C01349=1129.626,328.744,-79.221,-177.563,10.731,149.517
C01350=1129.630,328.496,-79.188,-177.566,10.728,149.517
C01351=1129.635,328.248,-79.155,-177.569,10.725,149.517
C01352=1129.638,328.001,-79.121,-177.573,10.723,149.517
C01353=1129.643,327.752,-79.087,-177.576,10.720,149.517
C01354=1129.647,327.505,-79.054,-177.579,10.718,149.518
C01355=1129.651,327.258,-79.020,-177.582,10.715,149.518
C01356=1129.655,327.010,-78.987,-177.586,10.713,149.518
C01357=1129.659,326.762,-78.954,-177.589,10.710,149.518
C01358=1129.662,326.514,-78.919,-177.592,10.708,149.518
C01359=1129.666,326.267,-78.886,-177.595,10.705,149.519
C01360=1129.670,326.019,-78.853,-177.598,10.702,149.519
C01361=1129.675,325.771,-78.820,-177.601,10.701,149.519
C01362=1129.678,325.524,-78.786,-177.604,10.698,149.519
C01363=1129.682,325.276,-78.753,-177.607,10.696,149.519
C01364=1129.686,325.028,-78.719,-177.610,10.693,149.520
C01365=1129.690,324.780,-78.686,-177.614,10.691,149.520
C01366=1129.694,324.532,-78.653,-177.617,10.688,149.520
C01367=1129.698,324.285,-78.620,-177.620,10.685,149.520
C01368=1129.702,324.038,-78.586,-177.623,10.683,149.520
C01369=1129.706,323.790,-78.553,-177.626,10.680,149.520
C01370=1129.711,323.542,-78.520,-177.630,10.678,149.521
C01371=1129.714,323.294,-78.486,-177.633,10.675,149.521
C01372=1129.718,323.046,-78.453,-177.636,10.673,149.521
C01373=1129.722,322.798,-78.420,-177.639,10.670,149.521
C01374=1129.727,322.551,-78.387,-177.642,10.668,149.521
C01375=1129.731,322.303,-78.354,-177.645,10.665,149.522
C01376=1129.734,322.090,-78.325,-177.648,10.663,149.522
C01377=1129.738,321.876,-78.297,-177.651,10.660,149.522
C01378=1129.741,321.664,-78.268,-177.654,10.659,149.522
C01379=1129.744,321.450,-78.240,-177.656,10.657,149.522
C01380=1129.748,321.237,-78.211,-177.659,10.654,149.523
C01381=1129.751,321.024,-78.182,-177.662,10.652,149.523
C01382=1129.755,320.810,-78.154,-177.665,10.650,149.523
C01383=1129.758,320.598,-78.125,-177.667,10.648,149.523
C01384=1129.762,320.349,-78.093,-177.671,10.645,149.523
C01385=1129.766,320.102,-78.060,-177.674,10.643,149.523
C01386=1129.770,319.854,-78.027,-177.677,10.640,149.524
C01387=1129.775,319.606,-77.994,-177.680,10.637,149.524
C01388=1129.779,319.359,-77.960,-177.683,10.635,149.524
C01389=1129.782,319.111,-77.928,-177.686,10.633,149.524
C01390=1129.786,318.863,-77.895,-177.689,10.630,149.524
C01391=1129.790,318.616,-77.862,-177.693,10.627,149.524
C01392=1129.795,318.367,-77.829,-177.696,10.625,149.525
C01393=1129.799,318.120,-77.796,-177.698,10.623,149.525
C01394=1129.802,317.872,-77.763,-177.702,10.621,149.525
C01395=1129.807,317.624,-77.730,-177.705,10.618,149.525
C01396=1129.811,317.376,-77.698,-177.708,10.615,149.525
C01397=1129.815,317.128,-77.665,-177.711,10.613,149.526
C01398=1129.818,316.881,-77.632,-177.714,10.610,149.526
C01399=1129.823,316.633,-77.599,-177.717,10.608,149.526
C01400=1129.827,316.385,-77.566,-177.721,10.605,149.526
C01401=1129.830,316.137,-77.534,-177.724,10.602,149.526
C01402=1129.835,315.890,-77.501,-177.727,10.600,149.526
C01403=1129.839,315.641,-77.468,-177.730,10.598,149.527
C01404=1129.843,315.394,-77.435,-177.733,10.595,149.527
C01405=1129.847,315.146,-77.403,-177.737,10.592,149.527
C01406=1129.851,314.898,-77.370,-177.740,10.590,149.527
C01407=1129.855,314.650,-77.337,-177.743,10.587,149.527
C01408=1129.859,314.402,-77.305,-177.746,10.585,149.528
C01409=1129.863,314.154,-77.272,-177.749,10.582,149.528
C01410=1129.867,313.906,-77.240,-177.752,10.579,149.528
C01411=1129.871,313.659,-77.207,-177.755,10.577,149.528
C01412=1129.875,313.410,-77.175,-177.758,10.575,149.528
C01413=1129.879,313.164,-77.142,-177.761,10.573,149.529
C01414=1129.883,312.916,-77.109,-177.764,10.570,149.529
C01415=1129.887,312.668,-77.077,-177.768,10.567,149.529
C01416=1129.892,312.419,-77.045,-177.771,10.565,149.529
C01417=1129.896,312.172,-77.012,-177.774,10.562,149.529
C01418=1129.899,311.924,-76.980,-177.777,10.560,149.530
C01419=1129.904,311.676,-76.947,-177.780,10.557,149.530
C01420=1129.907,311.428,-76.915,-177.784,10.555,149.530
C01421=1129.912,311.181,-76.882,-177.786,10.552,149.530
C01422=1129.916,310.933,-76.850,-177.790,10.549,149.530
C01423=1129.920,310.684,-76.818,-177.793,10.547,149.530
C01424=1129.924,310.437,-76.785,-177.796,10.544,149.531
C01425=1129.928,310.189,-76.753,-177.799,10.542,149.531
C01426=1129.932,309.941,-76.721,-177.802,10.539,149.531
C01427=1129.936,309.694,-76.688,-177.805,10.537,149.531
C01428=1129.940,309.446,-76.656,-177.808,10.535,149.531
C01429=1129.945,309.197,-76.624,-177.811,10.532,149.531
C01430=1129.948,308.949,-76.592,-177.815,10.530,149.532
C01431=1129.952,308.701,-76.559,-177.818,10.527,149.532
C01432=1129.956,308.489,-76.532,-177.820,10.524,149.532
C01433=1129.960,308.275,-76.504,-177.823,10.522,149.532
C01434=1129.963,308.062,-76.477,-177.825,10.520,149.532
C01435=1129.966,307.848,-76.449,-177.829,10.518,149.533
C01436=1129.970,307.635,-76.421,-177.831,10.516,149.533
C01437=1129.973,307.422,-76.393,-177.834,10.513,149.533
C01438=1129.977,307.208,-76.365,-177.837,10.512,149.533
C01439=1129.981,306.994,-76.338,-177.839,10.510,149.533
C01440=1129.985,306.747,-76.306,-177.842,10.507,149.533
C01441=1129.989,306.499,-76.274,-177.845,10.504,149.533
C01442=1129.993,306.251,-76.242,-177.849,10.502,149.534
C01443=1129.997,306.003,-76.209,-177.852,10.499,149.534
C01444=1130.002,305.756,-76.178,-177.855,10.497,149.534
C01445=1130.005,305.508,-76.146,-177.858,10.494,149.534
C01446=1130.010,305.259,-76.114,-177.861,10.492,149.534
C01447=1130.014,305.012,-76.082,-177.864,10.489,149.534
C01448=1130.018,304.764,-76.050,-177.867,10.486,149.535
C01449=1130.022,304.516,-76.018,-177.870,10.484,149.535
C01450=1130.026,304.267,-75.986,-177.874,10.481,149.535
C01451=1130.030,304.020,-75.955,-177.877,10.478,149.535
C01452=1130.035,303.772,-75.922,-177.879,10.477,149.535
C01453=1130.038,303.524,-75.890,-177.883,10.474,149.536
C01454=1130.043,303.276,-75.859,-177.886,10.472,149.536
C01455=1130.046,303.028,-75.827,-177.889,10.469,149.536
C01456=1130.051,302.780,-75.795,-177.892,10.466,149.536
C01457=1130.055,302.533,-75.763,-177.895,10.464,149.536
C01458=1130.059,302.285,-75.731,-177.898,10.461,149.537
C01459=1130.062,302.037,-75.699,-177.901,10.459,149.537
C01460=1130.068,301.788,-75.668,-177.904,10.456,149.537
C01461=1130.072,301.540,-75.636,-177.908,10.454,149.537
C01462=1130.076,301.293,-75.605,-177.911,10.451,149.537
C01463=1130.080,301.045,-75.573,-177.914,10.448,149.537
C01464=1130.083,300.797,-75.541,-177.917,10.446,149.538
C01465=1130.088,300.549,-75.510,-177.920,10.443,149.538
C01466=1130.092,300.301,-75.478,-177.923,10.441,149.538
C01467=1130.097,300.053,-75.446,-177.926,10.439,149.538
C01468=1130.100,299.805,-75.414,-177.929,10.436,149.538
C01469=1130.104,299.557,-75.383,-177.932,10.434,149.539
C01470=1130.109,299.309,-75.352,-177.935,10.431,149.539
C01471=1130.112,299.061,-75.320,-177.938,10.428,149.539
C01472=1130.117,298.814,-75.289,-177.941,10.426,149.539
C01473=1130.121,298.565,-75.257,-177.945,10.423,149.539
C01474=1130.124,298.317,-75.226,-177.948,10.420,149.539
C01475=1130.129,298.069,-75.193,-177.951,10.418,149.540
C01476=1130.133,297.821,-75.162,-177.954,10.415,149.540
C01477=1130.138,297.573,-75.131,-177.957,10.413,149.540
C01478=1130.142,297.325,-75.100,-177.961,10.410,149.540
C01479=1130.146,297.077,-75.068,-177.963,10.408,149.540
C01480=1130.150,296.829,-75.036,-177.966,10.406,149.540
C01481=1130.154,296.581,-75.006,-177.969,10.403,149.541
C01482=1130.158,296.333,-74.974,-177.972,10.400,149.541
C01483=1130.163,296.085,-74.943,-177.975,10.398,149.541
C01484=1130.166,295.837,-74.911,-177.978,10.395,149.541
C01485=1130.170,295.589,-74.880,-177.982,10.393,149.541
C01486=1130.175,295.341,-74.849,-177.985,10.390,149.542
C01487=1130.179,295.093,-74.817,-177.988,10.388,149.542
C01488=1130.183,294.880,-74.791,-177.990,10.386,149.542
C01489=1130.186,294.666,-74.763,-177.994,10.383,149.542
C01490=1130.189,294.453,-74.737,-177.996,10.381,149.542
C01491=1130.193,294.240,-74.710,-177.998,10.379,149.542
C01492=1130.197,294.026,-74.683,-178.001,10.376,149.542
C01493=1130.200,293.812,-74.656,-178.004,10.375,149.543
C01494=1130.204,293.599,-74.630,-178.006,10.373,149.543
C01495=1130.207,293.386,-74.602,-178.009,10.370,149.543
C01496=1130.212,293.138,-74.571,-178.012,10.368,149.543
C01497=1130.216,292.889,-74.540,-178.015,10.365,149.543
C01498=1130.219,292.642,-74.509,-178.019,10.362,149.544
C01499=1130.223,292.393,-74.478,-178.022,10.360,149.544
C01500=1130.228,292.145,-74.448,-178.024,10.358,149.544
C01501=1130.232,291.897,-74.416,-178.027,10.355,149.544
C01502=1130.236,291.649,-74.385,-178.030,10.352,149.544
C01503=1130.241,291.401,-74.354,-178.034,10.350,149.544
C01504=1130.244,291.153,-74.324,-178.036,10.347,149.545
C01505=1130.248,290.906,-74.292,-178.040,10.345,149.545
C01506=1130.252,290.657,-74.261,-178.043,10.342,149.545
C01507=1130.257,290.409,-74.230,-178.046,10.340,149.545
C01508=1130.261,290.160,-74.199,-178.049,10.337,149.545
C01509=1130.265,289.913,-74.169,-178.052,10.334,149.546
C01510=1130.269,289.665,-74.138,-178.055,10.332,149.546
C01511=1130.273,289.417,-74.106,-178.058,10.330,149.546
C01512=1130.278,289.169,-74.076,-178.061,10.327,149.546
C01513=1130.282,288.921,-74.045,-178.064,10.325,149.546
C01514=1130.286,288.673,-74.014,-178.067,10.322,149.546
C01515=1130.290,288.425,-73.984,-178.070,10.319,149.546
C01516=1130.295,288.177,-73.953,-178.073,10.317,149.547
C01517=1130.298,287.928,-73.922,-178.076,10.314,149.547
C01518=1130.303,287.681,-73.891,-178.080,10.312,149.547
C01519=1130.307,287.432,-73.860,-178.083,10.309,149.547
C01520=1130.310,287.185,-73.829,-178.086,10.307,149.548
C01521=1130.315,286.937,-73.799,-178.089,10.304,149.548
C01522=1130.320,286.689,-73.768,-178.092,10.302,149.548
C01523=1130.323,286.440,-73.737,-178.095,10.299,149.548
C01524=1130.328,286.192,-73.707,-178.098,10.297,149.548
C01525=1130.332,285.944,-73.676,-178.101,10.294,149.548
C01526=1130.336,285.695,-73.646,-178.104,10.291,149.548
C01527=1130.340,285.448,-73.615,-178.107,10.289,149.549
C01528=1130.344,285.200,-73.585,-178.110,10.286,149.549
C01529=1130.348,284.951,-73.554,-178.113,10.284,149.549
C01530=1130.353,284.703,-73.523,-178.116,10.281,149.549
C01531=1130.357,284.456,-73.493,-178.120,10.279,149.549
C01532=1130.361,284.208,-73.462,-178.123,10.276,149.550
C01533=1130.365,283.959,-73.432,-178.125,10.274,149.550
C01534=1130.369,283.711,-73.401,-178.128,10.272,149.550
C01535=1130.374,283.463,-73.371,-178.131,10.269,149.550
C01536=1130.378,283.215,-73.341,-178.135,10.266,149.550
C01537=1130.382,282.966,-73.310,-178.138,10.264,149.550
C01538=1130.386,282.719,-73.280,-178.141,10.261,149.551
C01539=1130.391,282.471,-73.249,-178.144,10.258,149.551
C01540=1130.395,282.223,-73.219,-178.147,10.256,149.551
C01541=1130.399,281.975,-73.189,-178.150,10.253,149.551
C01542=1130.403,281.726,-73.158,-178.153,10.250,149.551
C01543=1130.408,281.478,-73.128,-178.156,10.249,149.552
C01544=1130.411,281.265,-73.102,-178.159,10.246,149.552
C01545=1130.414,281.050,-73.076,-178.162,10.244,149.552
C01546=1130.418,280.837,-73.049,-178.165,10.241,149.552
C01547=1130.421,280.623,-73.024,-178.168,10.239,149.552
C01548=1130.425,280.410,-72.997,-178.171,10.236,149.552
C01549=1130.429,280.197,-72.972,-178.175,10.233,149.553
C01550=1130.432,279.983,-72.945,-178.177,10.231,149.553
C01551=1130.437,279.769,-72.920,-178.180,10.229,149.553
C01552=1130.441,279.521,-72.889,-178.184,10.225,149.553
C01553=1130.444,279.273,-72.860,-178.187,10.223,149.554
C01554=1130.449,279.025,-72.829,-178.190,10.221,149.554
C01555=1130.453,278.776,-72.799,-178.194,10.217,149.554
C01556=1130.458,278.528,-72.769,-178.197,10.215,149.554
C01557=1130.461,278.281,-72.738,-178.201,10.211,149.554
C01558=1130.466,278.032,-72.709,-178.204,10.209,149.555
C01559=1130.471,277.784,-72.679,-178.207,10.206,149.555
C01560=1130.474,277.535,-72.648,-178.211,10.204,149.555
C01561=1130.478,277.287,-72.619,-178.214,10.200,149.555
C01562=1130.482,277.040,-72.589,-178.218,10.198,149.555
C01563=1130.487,276.791,-72.559,-178.220,10.195,149.555
C01564=1130.491,276.543,-72.529,-178.224,10.192,149.556
C01565=1130.495,276.295,-72.499,-178.227,10.189,149.556
C01566=1130.500,276.046,-72.469,-178.230,10.186,149.556
C01567=1130.504,275.799,-72.439,-178.234,10.184,149.556
C01568=1130.508,275.551,-72.409,-178.237,10.181,149.556
C01569=1130.512,275.302,-72.380,-178.240,10.178,149.556
C01570=1130.516,275.055,-72.350,-178.243,10.176,149.557
C01571=1130.521,274.806,-72.320,-178.246,10.173,149.557
C01572=1130.525,274.558,-72.290,-178.249,10.169,149.557
C01573=1130.528,274.309,-72.260,-178.252,10.167,149.557
C01574=1130.532,274.061,-72.230,-178.256,10.164,149.557
C01575=1130.537,273.813,-72.201,-178.259,10.162,149.557
C01576=1130.542,273.564,-72.171,-178.262,10.159,149.557
C01577=1130.545,273.317,-72.141,-178.265,10.156,149.558
C01578=1130.550,273.068,-72.111,-178.267,10.153,149.558
C01579=1130.554,272.820,-72.082,-178.270,10.150,149.558
C01580=1130.558,272.572,-72.052,-178.274,10.148,149.558
C01581=1130.562,272.324,-72.023,-178.276,10.146,149.558
C01582=1130.566,272.076,-71.993,-178.279,10.143,149.558
C01583=1130.571,271.827,-71.963,-178.282,10.141,149.558
C01584=1130.575,271.579,-71.933,-178.285,10.138,149.558
C01585=1130.579,271.331,-71.904,-178.288,10.135,149.559
C01586=1130.584,271.083,-71.875,-178.291,10.132,149.559
C01587=1130.588,270.835,-71.845,-178.294,10.130,149.559
C01588=1130.592,270.587,-71.816,-178.296,10.128,149.559
C01589=1130.597,270.339,-71.786,-178.299,10.125,149.559
C01590=1130.601,270.090,-71.757,-178.302,10.122,149.559
C01591=1130.605,269.842,-71.727,-178.305,10.119,149.559
C01592=1130.609,269.594,-71.698,-178.307,10.117,149.559
C01593=1130.613,269.345,-71.668,-178.310,10.115,149.559
C01594=1130.618,269.097,-71.639,-178.313,10.112,149.559
C01595=1130.622,268.849,-71.610,-178.315,10.110,149.560
C01596=1130.626,268.601,-71.580,-178.318,10.107,149.560
C01597=1130.630,268.352,-71.551,-178.321,10.105,149.560
C01598=1130.634,268.104,-71.521,-178.323,10.102,149.560
C01599=1130.638,267.856,-71.492,-178.326,10.099,149.560
C01600=1130.642,267.642,-71.467,-178.328,10.097,149.560
C01601=1130.646,267.429,-71.441,-178.331,10.095,149.560
C01602=1130.650,267.215,-71.416,-178.333,10.093,149.560
C01603=1130.654,267.001,-71.391,-178.335,10.091,149.560
C01604=1130.657,266.787,-71.366,-178.337,10.089,149.560
C01605=1130.661,266.573,-71.340,-178.339,10.087,149.560
C01606=1130.665,266.359,-71.315,-178.342,10.085,149.561
C01607=1130.668,266.146,-71.290,-178.344,10.083,149.560
C01608=1130.673,265.898,-71.261,-178.346,10.081,149.561
C01609=1130.677,265.649,-71.231,-178.348,10.079,149.561
C01610=1130.681,265.401,-71.202,-178.351,10.076,149.561
C01611=1130.686,265.152,-71.173,-178.354,10.074,149.561
C01612=1130.690,264.905,-71.145,-178.356,10.072,149.561
C01613=1130.694,264.657,-71.115,-178.358,10.069,149.561
C01614=1130.698,264.408,-71.086,-178.361,10.067,149.561
C01615=1130.702,264.160,-71.056,-178.365,10.064,149.561
C01616=1130.707,263.911,-71.027,-178.369,10.061,149.562
C01617=1130.711,263.664,-70.998,-178.373,10.057,149.562
C01618=1130.716,263.415,-70.969,-178.377,10.054,149.562
C01619=1130.719,263.167,-70.941,-178.381,10.051,149.563
C01620=1130.723,262.919,-70.911,-178.385,10.048,149.563
C01621=1130.728,262.670,-70.882,-178.388,10.044,149.563
C01622=1130.733,262.422,-70.853,-178.392,10.041,149.563
C01623=1130.737,262.174,-70.824,-178.396,10.039,149.564
C01624=1130.741,261.925,-70.796,-178.399,10.035,149.564
C01625=1130.745,261.677,-70.766,-178.403,10.032,149.564
C01626=1130.750,261.429,-70.737,-178.406,10.029,149.564
C01627=1130.754,261.181,-70.709,-178.410,10.026,149.564
C01628=1130.758,260.933,-70.680,-178.414,10.023,149.564
C01629=1130.762,260.684,-70.651,-178.417,10.020,149.564
C01630=1130.767,260.436,-70.622,-178.421,10.017,149.565
C01631=1130.771,260.188,-70.594,-178.423,10.014,149.565
C01632=1130.775,259.939,-70.564,-178.427,10.010,149.565
C01633=1130.779,259.690,-70.536,-178.430,10.008,149.565
C01634=1130.784,259.443,-70.508,-178.434,10.004,149.565
C01635=1130.788,259.194,-70.478,-178.437,10.002,149.565
C01636=1130.792,258.945,-70.450,-178.440,9.998,149.566
C01637=1130.796,258.698,-70.421,-178.443,9.995,149.566
C01638=1130.801,258.449,-70.392,-178.446,9.993,149.566
C01639=1130.805,258.200,-70.364,-178.450,9.989,149.566
C01640=1130.809,257.953,-70.335,-178.453,9.986,149.566
C01641=1130.814,257.704,-70.306,-178.456,9.984,149.566
C01642=1130.818,257.456,-70.278,-178.459,9.981,149.566
C01643=1130.822,257.208,-70.249,-178.462,9.977,149.566
C01644=1130.827,256.959,-70.220,-178.465,9.975,149.566
C01645=1130.831,256.711,-70.192,-178.468,9.972,149.567
C01646=1130.836,256.462,-70.164,-178.471,9.969,149.567
C01647=1130.839,256.214,-70.135,-178.474,9.966,149.567
C01648=1130.844,255.966,-70.107,-178.477,9.964,149.567
C01649=1130.848,255.718,-70.079,-178.476,9.963,149.566
C01650=1130.852,255.469,-70.050,-178.475,9.962,149.566
C01651=1130.856,255.222,-70.021,-178.475,9.961,149.566
C01652=1130.861,254.973,-69.993,-178.474,9.961,149.565
C01653=1130.865,254.724,-69.964,-178.474,9.960,149.565
C01654=1130.870,254.476,-69.936,-178.475,9.959,149.565
C01655=1130.874,254.227,-69.908,-178.475,9.958,149.565
C01656=1130.877,254.014,-69.883,-178.476,9.956,149.565
C01657=1130.881,253.800,-69.858,-178.477,9.955,149.565
C01658=1130.885,253.586,-69.834,-178.478,9.954,149.565
C01659=1130.889,253.372,-69.809,-178.479,9.952,149.565
C01660=1130.893,253.158,-69.785,-178.480,9.951,149.565
C01661=1130.895,252.945,-69.760,-178.482,9.949,149.565
C01662=1130.899,252.731,-69.736,-178.484,9.947,149.565
C01663=1130.903,252.517,-69.711,-178.486,9.946,149.565
C01664=1130.908,252.268,-69.683,-178.489,9.943,149.565
C01665=1130.912,252.020,-69.655,-178.492,9.940,149.565
C01666=1130.917,251.771,-69.626,-178.495,9.938,149.565
C01667=1130.921,251.523,-69.598,-178.498,9.936,149.566
C01668=1130.925,251.274,-69.570,-178.502,9.932,149.566
C01669=1130.929,251.027,-69.541,-178.506,9.929,149.566
C01670=1130.933,250.778,-69.513,-178.510,9.926,149.567
C01671=1130.938,250.530,-69.485,-178.514,9.923,149.567
C01672=1130.942,250.281,-69.456,-178.519,9.919,149.567
C01673=1130.946,250.034,-69.429,-178.524,9.915,149.568
C01674=1130.951,249.785,-69.400,-178.530,9.911,149.568
C01675=1130.955,249.537,-69.372,-178.535,9.907,149.569
C01676=1130.959,249.288,-69.344,-178.541,9.902,149.569
C01677=1130.964,249.039,-69.316,-178.547,9.898,149.569
C01678=1130.968,248.791,-69.288,-178.553,9.893,149.570
C01679=1130.972,248.543,-69.260,-178.560,9.888,149.571
C01680=1130.977,248.294,-69.232,-178.566,9.883,149.571
C01681=1130.981,248.046,-69.204,-178.574,9.878,149.572
C01682=1130.985,247.798,-69.176,-178.581,9.872,149.572
C01683=1130.990,247.549,-69.149,-178.588,9.867,149.573
C01684=1130.994,247.300,-69.120,-178.593,9.862,149.573
C01685=1130.999,247.052,-69.092,-178.594,9.861,149.573
C01686=1131.003,246.804,-69.065,-178.595,9.858,149.573
C01687=1131.007,246.555,-69.037,-178.596,9.856,149.573
C01688=1131.011,246.307,-69.009,-178.597,9.854,149.572
C01689=1131.015,246.058,-68.982,-178.599,9.852,149.572
C01690=1131.020,245.810,-68.953,-178.600,9.850,149.572
C01691=1131.025,245.562,-68.926,-178.601,9.848,149.572
C01692=1131.029,245.313,-68.898,-178.603,9.846,149.572
C01693=1131.033,245.065,-68.870,-178.604,9.844,149.572
C01694=1131.038,244.817,-68.843,-178.605,9.841,149.571
C01695=1131.042,244.568,-68.815,-178.607,9.839,149.571
C01696=1131.046,244.320,-68.787,-178.609,9.838,149.571
C01697=1131.051,244.071,-68.759,-178.610,9.835,149.571
C01698=1131.055,243.823,-68.732,-178.612,9.834,149.571
C01699=1131.060,243.574,-68.705,-178.613,9.831,149.571
C01700=1131.063,243.326,-68.676,-178.615,9.829,149.571
C01701=1131.068,243.077,-68.649,-178.617,9.826,149.571
C01702=1131.072,242.829,-68.622,-178.619,9.824,149.571
C01703=1131.076,242.581,-68.593,-178.620,9.822,149.571
C01704=1131.081,242.332,-68.566,-178.622,9.820,149.571
C01705=1131.085,242.084,-68.539,-178.624,9.818,149.571
C01706=1131.089,241.835,-68.511,-178.626,9.816,149.571
C01707=1131.094,241.587,-68.483,-178.628,9.813,149.571
C01708=1131.098,241.339,-68.456,-178.630,9.811,149.571
C01709=1131.102,241.090,-68.428,-178.632,9.809,149.571
C01710=1131.107,240.842,-68.401,-178.635,9.806,149.571
C01711=1131.112,240.593,-68.374,-178.637,9.804,149.571
C01712=1131.115,240.379,-68.350,-178.638,9.802,149.571
C01713=1131.119,240.165,-68.327,-178.640,9.800,149.571
C01714=1131.123,239.951,-68.302,-178.642,9.798,149.571
C01715=1131.127,239.737,-68.279,-178.645,9.796,149.571
C01716=1131.130,239.523,-68.255,-178.646,9.794,149.571
C01717=1131.134,239.309,-68.232,-178.649,9.792,149.571
C01718=1131.137,239.095,-68.208,-178.651,9.789,149.571
C01719=1131.142,238.881,-68.184,-178.653,9.787,149.571
C01720=1131.146,238.633,-68.156,-178.655,9.785,149.571
C01721=1131.150,238.384,-68.129,-178.658,9.782,149.571
C01722=1131.155,238.136,-68.102,-178.660,9.780,149.571
C01723=1131.159,237.888,-68.074,-178.663,9.777,149.571
C01724=1131.163,237.638,-68.047,-178.666,9.774,149.571
C01725=1131.168,237.390,-68.020,-178.668,9.772,149.571
C01726=1131.172,237.142,-67.992,-178.671,9.770,149.572
C01727=1131.176,236.894,-67.966,-178.674,9.767,149.572
C01728=1131.180,236.645,-67.938,-178.677,9.764,149.572
C01729=1131.185,236.396,-67.911,-178.679,9.762,149.572
C01730=1131.189,236.148,-67.883,-178.682,9.759,149.572
C01731=1131.194,235.900,-67.856,-178.685,9.756,149.572
C01732=1131.199,235.651,-67.829,-178.687,9.754,149.572
C01733=1131.203,235.402,-67.802,-178.690,9.751,149.572
C01734=1131.207,235.154,-67.775,-178.693,9.748,149.572
C01735=1131.211,234.906,-67.748,-178.697,9.745,149.573
C01736=1131.216,234.658,-67.720,-178.700,9.742,149.573
C01737=1131.220,234.408,-67.693,-178.703,9.739,149.573
C01738=1131.224,234.160,-67.666,-178.706,9.737,149.573
C01739=1131.229,233.911,-67.639,-178.710,9.733,149.573
C01740=1131.234,233.663,-67.612,-178.713,9.730,149.573
C01741=1131.238,233.415,-67.585,-178.716,9.728,149.573
C01742=1131.242,233.166,-67.558,-178.719,9.724,149.574
C01743=1131.246,232.917,-67.531,-178.722,9.721,149.574
C01744=1131.251,232.669,-67.504,-178.726,9.718,149.574
C01745=1131.255,232.421,-67.477,-178.729,9.715,149.574
C01746=1131.259,232.172,-67.450,-178.733,9.712,149.574
C01747=1131.264,231.924,-67.423,-178.736,9.708,149.574
C01748=1131.269,231.675,-67.396,-178.740,9.705,149.574
C01749=1131.273,231.427,-67.370,-178.743,9.703,149.575
C01750=1131.277,231.178,-67.343,-178.747,9.699,149.575
C01751=1131.282,230.930,-67.316,-178.750,9.695,149.575
C01752=1131.285,230.681,-67.289,-178.754,9.692,149.575
C01753=1131.290,230.432,-67.262,-178.758,9.689,149.575
C01754=1131.295,230.184,-67.235,-178.762,9.685,149.576
C01755=1131.299,229.936,-67.208,-178.766,9.682,149.576
C01756=1131.303,229.687,-67.181,-178.770,9.678,149.576
C01757=1131.308,229.438,-67.155,-178.773,9.674,149.576
C01758=1131.312,229.190,-67.128,-178.777,9.671,149.576
C01759=1131.317,228.941,-67.101,-178.781,9.668,149.577
C01760=1131.321,228.693,-67.075,-178.785,9.664,149.577
C01761=1131.325,228.445,-67.048,-178.788,9.661,149.577
C01762=1131.330,228.196,-67.022,-178.792,9.657,149.577
C01763=1131.334,227.947,-66.995,-178.795,9.654,149.577
C01764=1131.338,227.699,-66.968,-178.799,9.650,149.577
C01765=1131.343,227.450,-66.942,-178.802,9.646,149.577
C01766=1131.348,227.202,-66.915,-178.806,9.643,149.577
C01767=1131.352,226.953,-66.889,-178.810,9.639,149.577
C01768=1131.355,226.738,-66.866,-178.813,9.637,149.578
C01769=1131.359,226.525,-66.843,-178.815,9.634,149.578
C01770=1131.363,226.310,-66.820,-178.818,9.631,149.578
C01771=1131.367,226.097,-66.797,-178.822,9.627,149.578
C01772=1131.371,225.882,-66.775,-178.824,9.624,149.578
C01773=1131.375,225.668,-66.752,-178.827,9.621,149.578
C01774=1131.379,225.454,-66.729,-178.830,9.618,149.578
C01775=1131.382,225.240,-66.706,-178.833,9.616,149.578
C01776=1131.386,224.991,-66.680,-178.836,9.612,149.578
C01777=1131.391,224.743,-66.653,-178.839,9.609,149.578
C01778=1131.395,224.494,-66.628,-178.842,9.605,149.578
C01779=1131.399,224.246,-66.601,-178.845,9.602,149.578
C01780=1131.404,223.997,-66.575,-178.848,9.598,149.578
C01781=1131.409,223.749,-66.549,-178.851,9.596,149.578
C01782=1131.414,223.500,-66.522,-178.854,9.592,149.578
C01783=1131.418,223.251,-66.497,-178.857,9.589,149.578
C01784=1131.422,223.003,-66.470,-178.860,9.585,149.578
C01785=1131.427,222.754,-66.444,-178.863,9.582,149.578
